(* CoDeSys 2.3.9.50 project: WTP_Pro_15_8_2016.pro *)
(* Libraries: STANDARD.LIB 5.6.98 12:03:02 *)

(* Task configuration *)
TASK Standard (PRIORITY := 0, INTERVAL := T#500ms);
	MAIN
END_TASK

(* Global variable list: Global_Variables *)
VAR_GLOBAL
	dummy: BOOL;
	GlobalON: TIME := T#5s;
	GlobalOFF: TIME := T#5s;
END_VAR

(* Data type *)
TYPE TEST :
STRUCT
	x : POINTER TO BOOL;
END_STRUCT
END_TYPE

(* Data type *)
TYPE TEST2 :
STRUCT
	X : BOOL;
END_STRUCT
END_TYPE

(* POU MAIN, ST *)
PROGRAM MAIN
VAR
	fbINLET_NEW_A: INLET_NEW_A;
	fbREUSE_WATER: REUSE_WATER;
END_VAR
STREAM_INLET_MIXER_1;
STREAM_INLET_MIXER_2;
INLET_SCREENING_OPERATION_2;
GRIT_REMOVAL_OPERATION;
SBR_TRANSFER_1;
SBR_TRANSFER_2;
REUSE_WATER_SYSTEM;
SBR_REACTOR_1;
SBR_REACTOR_2;
SLUDGE_THICKENING;

fbINLET_NEW_A();
fbREUSE_WATER();
END_PROGRAM

(* POU INLET_NEW_A, ST *)
FUNCTION_BLOCK INLET_NEW_A
VAR_INPUT
(*inlet*)
	i1: BOOL;
	i3: BOOL;
	i2: BOOL;
	i4: BOOL;

(*MIXER*)

	i5: BOOL;
	i6: BOOL;

(*penstock*)
	r1: BOOL; (*rs1*)
	i7: BOOL; (*ps open*)
	i8: BOOL;	(*ps open*)
	i10: BOOL;
	i9: BOOL;
	i11: BOOL;
	s1: BOOL;
	s2: BOOL;
	s3: BOOL;
	s4: BOOL;

(* sbr transfer *)
	i12: BOOL;
	i13: BOOL;


END_VAR
VAR_OUTPUT

(*inlet*)
	q1: BOOL;
	q2: BOOL;

(*MIXER*)

	q3: BOOL;
	q4: BOOL;

(*penstock*)
	q5: BOOL; (*ps1*)
	q6: BOOL; (*ps2*)
	q7: BOOL;
	q8: BOOL;
	q10: BOOL;
	q9: BOOL;
	q11: BOOL;
	q12: BOOL;
	q13: BOOL;
	q14: BOOL;
	q15: BOOL;
	q16: BOOL;
	q17: BOOL;
	q18: BOOL;
	q19: BOOL;
	q20: BOOL;
(* Grit Removal*)

	q21: BOOL;
	q22: BOOL;
	q23: BOOL;
	q24: BOOL;
	q25:BOOL;
	q26:BOOL;

(* sbr transfer *)

	q27: BOOL;
	q28: BOOL;

END_VAR
VAR
(*inlet*)
	m1: BOOL;
	ton1: TON;

(*MIXER*)


(*penstock*)
	penstock: INT;
	FailedGroupA: BOOL;
	FailedGroupB: BOOL;
	m2: BOOL;
	TP1: TP;
	m3: BOOL;
	TON2: TON;
	TON3: TON;
	TOF1: TOF;
	TON4 : TON;
	mr: BOOL;
	F_TRIG1: F_TRIG;
	R_TRIG1: R_TRIG;
	m4 : BOOL;
	TON5: TON;

END_VAR



(*
CASE penstock OF
0:
	q5 := TRUE;
	q6 := FALSE;
	IF FailedGroupA OR m2 THEN
		penstock := 1;
	END_IF
1 :
 	q6 := TRUE;
	IF FailedGroupB THEN
		penstock := 2;
	ELSIF i8 THEN
		penstock := 3;
	END_IF
2 :
	q5 := FALSE;
	q6 := FALSE;
	IF r1 THEN
		penstock := 0;
	END_IF
3:
	q6 := TRUE;
	q5 := FALSE;
	IF FailedGroupB OR m2 THEN
		penstock := 4;
	END_IF
4 :
	q6 := TRUE;
	IF FailedGroupA THEN
		penstock := 2;
	ELSIF i7 THEN
		penstock := 0;
	END_IF
END_CASE*)
(*EQ Pump*)
q1 := NOT i1 OR i3 OR m1;
q2 := i2 AND NOT i3 AND NOT m1;
ton1(IN:=i4 , PT:=t#5m , Q=>m1 , ET=> );

(*Mixer*)
q3 := NOT i5;
q4 := i6;


(*screen*)
FailedGroupA := s1 OR s2;
FailedGroupB := s3 OR s4;

m4 := ((NOT m4 AND (FailedGroupA OR m2)) OR m4) AND NOT((m4 AND (FailedGroupB OR m2)) OR r1);
q5 := (NOT m4 OR q5) AND NOT(( m4 AND i8) OR mr) ;
q6 := (m4 OR q6) AND NOT ((NOT m4 AND i7) OR mr);
mr := (mr OR (FailedGroupA AND FailedGroupB)) AND NOT r1;

TOF1(IN:=i11 , PT:=T#2m , Q=>i9 , ET=> );

F_TRIG1(CLK:=m4 );
R_TRIG1(CLK:=m4 );
TP1(IN:=(F_TRIG1.Q OR R_TRIG1.Q) , PT:= T#5m , Q=>m3 , ET=> );
m2 := i10 AND NOT m3;

TON4(IN:=NOT i9 OR NOT(q5 OR q6) , PT:=T#5m , Q=>q7 , ET=> );
TON2(IN:= i9 AND (q5 OR q6), PT := T#1h, Q=> q8);

TON3(IN:=q7,PT:=T#5m,Q=>q9);
q10 := q8;

q11 := q9;
q12 := q10;

q13 := NOT (i9 AND Q5);
q14 := (i9 AND Q5);

q15 := NOT(i9 AND q6);
q16 := (i9 AND q6);

q17 := q13;
q18 := q14;

q19 := q15;
q20 :=q18;

(*Grit Removal*)
q21 := i7;
q22 := i8;

q23 := NOT i9;
q24 := i9;

TON5(IN:= NOT i9, PT:=T#5m , Q=>q25 );
q26 := i9;


(*sbr transfer*)
q27  := NOT i12;
q28 := i13;
END_FUNCTION_BLOCK

(* POU REUSE_WATER, ST *)
FUNCTION_BLOCK REUSE_WATER
VAR_INPUT
	i3: BOOL;
	i1: BOOL;
	i4: BOOL;
	i2: BOOL;
	i5: BOOL;
	a1 : INT;
END_VAR
VAR_OUTPUT
	q1: BOOL;
	q2: BOOL;
	q3: BOOL;
	q4: BOOL;
	q5: BOOL;
	q6: BOOL;
	q7: BOOL;
	q8: BOOL;
	q9: BOOL;
END_VAR
VAR
	m1: BOOL;
	e1: BOOL;
	p1: REAL;
	TON1: TON;
	m2: BOOL;
END_VAR
p1 := INT_TO_REAL(a1) * (20.0/32767.0);

q1 := (p1 > 8) OR (NOT m1) OR e1 OR i3;
q2 := (p1 <= 6) AND m1;

q3:=(p1 > 6.4) OR (NOT m1) OR e1 OR i3;
q4 := (p1 <= 5.2) AND m1;

q5:=(p1 > 5.9) OR (NOT m1) OR e1 OR i3;
q6 := (p1 <= 4.7) AND m1;

TON1(IN:=((p1 < 3.5) AND m1) , PT:=T#5s , Q=>e1 , ET=> );
m2 := (i2 OR m2) AND i1;
m1 := i4 AND m2;

q7 := NOT i5 OR q7;
q8 := i5 AND q8;

q9 := TRUE;
END_FUNCTION_BLOCK

(* POU STREAM_INLET_MIXER_1, CFC *)
PROGRAM STREAM_INLET_MIXER_1
VAR
	LSL101A : inBlock;
	LSS101A : inBlock;
	LSH101A : inBlock;
	LSD101A : inBlock;
	LSL100A : inBlock;
	LSHL100A:inBlock;

	bCriticalEQFloatHi: BOOL;
	bWarningFloatSensorLow: BOOL;
	bCriticalFloatSensorDry: BOOL;



	EQPump_P101A_1_remote_mode AT%I* : BOOL;
	EQPump_P101A_1_overload AT%I* : BOOL;
	EQPump_P101A_1_incomplete AT%I* : BOOL;
	EQPump_P101A_1_status AT%I* : BOOL;

	EQPump_P101A_1_command AT%Q* : BOOL;

	EQPump_P101A_1_in : BOOL;
	EQPump_P101A_1_overload_error : BOOL;
	EQPump_P101A_1_incomplete_error : BOOL;
	EQPump_P101A_1_status_error : BOOL;
	EQPump_P101A_1_common_error : BOOL;
	EQPump_P101A_1_stop_error : BOOL;

	EQPump_P101A_1_overload_Filter : ErrorFilter;
	EQPump_P101A_1_incomplete_Filter : ErrorFilter;
	EQPump_P101A_1_status_Filter : ErrorFilter;
	EQPump_P101A_1_stop_Filter : ErrorFilter;



	EQPump_P101A_2_remote_mode AT%I* : BOOL;
	EQPump_P101A_2_overload AT%I* : BOOL;
	EQPump_P101A_2_incomplete AT%I* : BOOL;
	EQPump_P101A_2_status AT%I* : BOOL;

	EQPump_P101A_2_command AT%Q* : BOOL;

	EQPump_P101A_2_in : BOOL;
	EQPump_P101A_2_overload_error : BOOL;
	EQPump_P101A_2_incomplete_error : BOOL;
	EQPump_P101A_2_status_error : BOOL;
	EQPump_P101A_2_common_error : BOOL;
	EQPump_P101A_2_stop_error : BOOL;

	EQPump_P101A_2_overload_Filter : ErrorFilter;
	EQPump_P101A_2_incomplete_Filter : ErrorFilter;
	EQPump_P101A_2_status_Filter : ErrorFilter;
	EQPump_P101A_2_stop_Filter : ErrorFilter;

	EQPump_P101A_CriticalStartError : BOOL;

	Mixer_M101A_1_remote_mode AT%I* : BOOL;
	Mixer_M101A_1_overload AT%I* : BOOL;
	Mixer_M101A_1_incomplete AT%I* : BOOL;
	Mixer_M101A_1_status AT%I* : BOOL;

	Mixer_M101A_1_command AT%Q* : BOOL;

	Mixer_M101A_1_in : BOOL;
	Mixer_M101A_1_overload_error : BOOL;
	Mixer_M101A_1_incomplete_error : BOOL;
	Mixer_M101A_1_status_error : BOOL;
	Mixer_M101A_1_common_error : BOOL;
	Mixer_M101A_1_stop_error : BOOL;


	Mixer_M101A_1_overload_Filter : ErrorFilter;
	Mixer_M101A_1_incomplete_Filter : ErrorFilter;
	Mixer_M101A_1_status_Filter : ErrorFilter;
	Mixer_M101A_1_stop_Filter : ErrorFilter;


	Mixer_M101A_2_remote_mode AT%I* : BOOL;
	Mixer_M101A_2_overload AT%I* : BOOL;
	Mixer_M101A_2_incomplete AT%I* : BOOL;
	Mixer_M101A_2_status AT%I* : BOOL;

	Mixer_M101A_2_command AT%Q* : BOOL;

	Mixer_M101A_2_in : BOOL;
	Mixer_M101A_2_overload_error : BOOL;
	Mixer_M101A_2_incomplete_error : BOOL;
	Mixer_M101A_2_status_error : BOOL;
	Mixer_M101A_2_common_error : BOOL;
	Mixer_M101A_2_stop_error : BOOL;

	Mixer_M101A_2_overload_Filter : ErrorFilter;
	Mixer_M101A_2_incomplete_Filter : ErrorFilter;
	Mixer_M101A_2_status_Filter : ErrorFilter;
	Mixer_M101A_2_stop_Filter : ErrorFilter;

	Mixer_M101A_CriticalStartEror : BOOL;

	InletPump :Equipment_Dual;
	Mixer :Equipment_Dual;



END_VAR
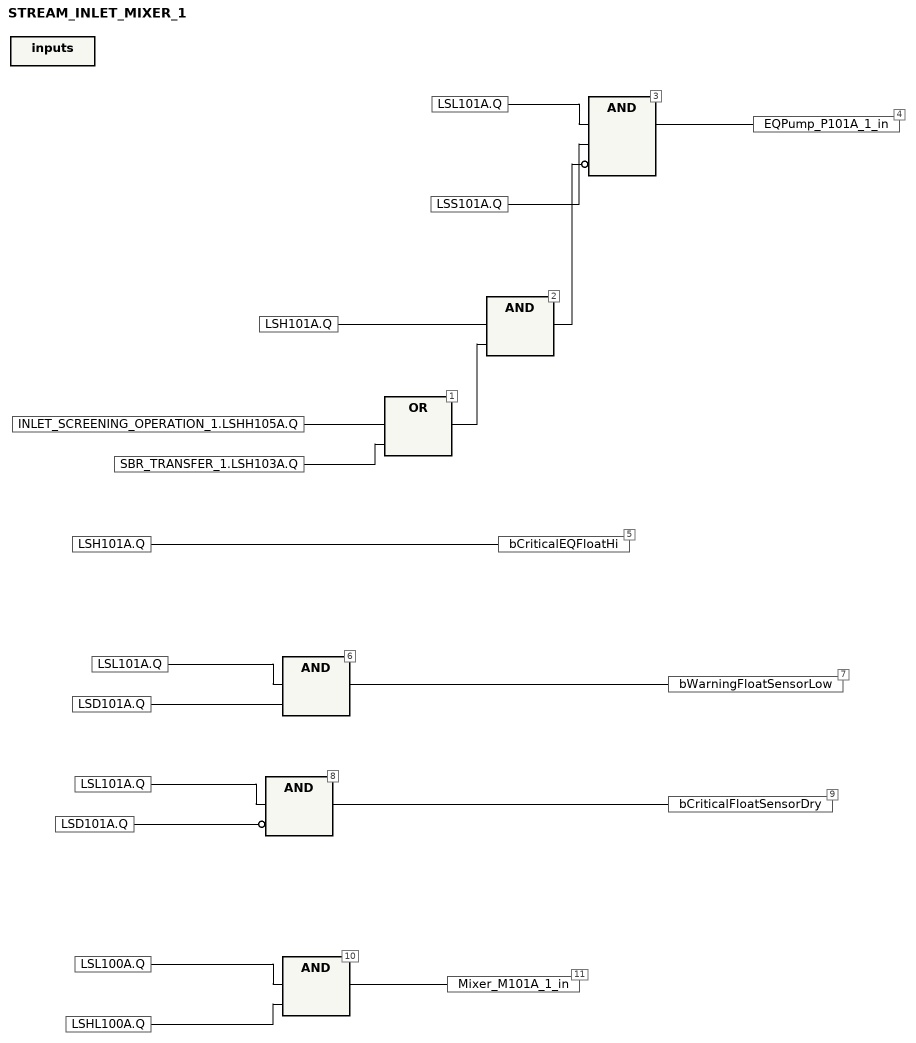
_CFC_ (* Continuous Function Chart, elements in execution order *)
#0 inputs()
#1 OR(INLET_SCREENING_OPERATION_1.LSHH105A.Q, SBR_TRANSFER_1.LSH103A.Q)
#2 AND(LSH101A.Q, #1)
#3 AND(LSL101A.Q, LSS101A.Q, NOT #2)
#4 EQPump_P101A_1_in <= #3
#5 bCriticalEQFloatHi <= LSH101A.Q
#6 AND(LSL101A.Q, LSD101A.Q)
#7 bWarningFloatSensorLow <= #6
#8 AND(LSL101A.Q, NOT LSD101A.Q)
#9 bCriticalFloatSensorDry <= #8
#10 AND(LSL100A.Q, LSHL100A.Q)
#11 Mixer_M101A_1_in <= #10
_END_CFC_
(* the same logic as Structured Text *)
inputs();
EQPump_P101A_1_in := LSL101A.Q AND LSS101A.Q AND NOT (LSH101A.Q AND (INLET_SCREENING_OPERATION_1.LSHH105A.Q OR SBR_TRANSFER_1.LSH103A.Q));
bCriticalEQFloatHi := LSH101A.Q;
bWarningFloatSensorLow := LSL101A.Q AND LSD101A.Q;
bCriticalFloatSensorDry := LSL101A.Q AND NOT LSD101A.Q;
Mixer_M101A_1_in := LSL100A.Q AND LSHL100A.Q;
END_PROGRAM
ACTION inputs:
	LSL101A();
	LSS101A();
	LSH101A();
	LSD101A();

	LSL100A();
	LSHL100A();



EQPump_P101A_1_overload_Filter(IN:=(EQPump_P101A_1_overload AND EQPump_P101A_1_in),PT:=T#10s,Q=>EQPump_P101A_1_overload_error);
EQPump_P101A_1_incomplete_Filter(IN:=(EQPump_P101A_1_incomplete AND EQPump_P101A_1_in),PT:=T#2s,Q=>EQPump_P101A_1_incomplete_error);
EQPump_P101A_1_status_Filter(IN:=(NOT EQPump_P101A_1_status AND EQPump_P101A_1_in),PT:=T#2s, Q=>EQPump_P101A_1_status_error);
EQPump_P101A_1_stop_Filter(IN:=( EQPump_P101A_1_status AND NOT EQPump_P101A_1_in),PT:=T#10s, Q=>EQPump_P101A_1_stop_error);

EQPump_P101A_1_common_error := EQPump_P101A_1_overload_error OR EQPump_P101A_1_incomplete_error OR EQPump_P101A_1_status_error OR EQPump_P101A_1_stop_error;



EQPump_P101A_2_overload_Filter(IN:=(EQPump_P101A_2_overload AND EQPump_P101A_2_in),PT:=T#10s,Q=>EQPump_P101A_2_overload_error);
EQPump_P101A_2_incomplete_Filter(IN:=(EQPump_P101A_2_incomplete AND EQPump_P101A_2_in),PT:=T#2s,Q=>EQPump_P101A_2_incomplete_error);
EQPump_P101A_2_status_Filter(IN:=(NOT EQPump_P101A_2_status AND EQPump_P101A_2_in),PT:=T#2s, Q=>EQPump_P101A_2_status_error);
EQPump_P101A_2_stop_Filter(IN:=( EQPump_P101A_2_status AND NOT EQPump_P101A_2_in),PT:=T#10s, Q=>EQPump_P101A_2_stop_error);

EQPump_P101A_2_common_error := EQPump_P101A_2_overload_error OR EQPump_P101A_2_incomplete_error OR EQPump_P101A_2_status_error OR EQPump_P101A_2_stop_error;

InletPump(
	ERROR1:=EQPump_P101A_1_common_error ,
	ERROR2:=EQPump_P101A_2_common_error ,
	IN1:=EQPump_P101A_1_in ,
	IN2:=EQPump_P101A_2_in ,
	remote1:=EQPump_P101A_1_remote_mode ,
	remote2:= EQPump_P101A_2_remote_mode,
	Command1=>EQPump_P101A_1_command ,
	Command2=>EQPump_P101A_2_command );


EQPump_P101A_CriticalStartError := EQPump_P101A_1_common_error AND EQPump_P101A_2_common_error;


Mixer_M101A_1_overload_Filter(IN:=(Mixer_M101A_1_overload AND Mixer_M101A_1_in),PT:=T#10s,Q=>Mixer_M101A_1_overload_error);
Mixer_M101A_1_incomplete_Filter(IN:=(Mixer_M101A_1_incomplete AND Mixer_M101A_1_in),PT:=T#2s,Q=>Mixer_M101A_1_incomplete_error);
Mixer_M101A_1_status_Filter(IN:=(NOT Mixer_M101A_1_status AND Mixer_M101A_1_in),PT:=T#2s, Q=>Mixer_M101A_1_status_error);
Mixer_M101A_1_stop_Filter(IN:=( Mixer_M101A_1_status AND NOT Mixer_M101A_1_in),PT:=T#10s, Q=>Mixer_M101A_1_stop_error);

Mixer_M101A_1_common_error := Mixer_M101A_1_overload_error OR Mixer_M101A_1_incomplete_error OR Mixer_M101A_1_status_error OR Mixer_M101A_1_stop_error;


Mixer_M101A_2_overload_Filter(IN:=(Mixer_M101A_2_overload AND Mixer_M101A_2_in),PT:=T#10s,Q=>Mixer_M101A_2_overload_error);
Mixer_M101A_2_incomplete_Filter(IN:=(Mixer_M101A_2_incomplete AND Mixer_M101A_2_in),PT:=T#2s,Q=>Mixer_M101A_2_incomplete_error);
Mixer_M101A_2_status_Filter(IN:=(NOT Mixer_M101A_2_status AND Mixer_M101A_2_in),PT:=T#2s, Q=>Mixer_M101A_2_status_error);
Mixer_M101A_2_stop_Filter(IN:=( Mixer_M101A_2_status AND NOT Mixer_M101A_2_in),PT:=T#10s, Q=>Mixer_M101A_2_stop_error);

Mixer_M101A_2_common_error := Mixer_M101A_2_overload_error OR Mixer_M101A_2_incomplete_error OR Mixer_M101A_2_status_error OR Mixer_M101A_2_stop_error;

Mixer(
	ERROR1:=Mixer_M101A_1_common_error ,
	ERROR2:=Mixer_M101A_2_common_error ,
	remote1:=Mixer_M101A_1_remote_mode ,
	remote2:= Mixer_M101A_2_remote_mode,
	IN1:=Mixer_M101A_1_in ,
	IN2:=Mixer_M101A_2_in ,
	Command1=>Mixer_M101A_1_command,
	Command2=>Mixer_M101A_2_command );

Mixer_M101A_CriticalStartEror := Mixer_M101A_1_common_error AND Mixer_M101A_2_common_error;
END_ACTION

(* POU module/inBlock, ST *)
FUNCTION_BLOCK inBlock
VAR_INPUT
END_VAR
VAR_OUTPUT
	Q : BOOL;
END_VAR
VAR
	IN AT%I* : BOOL;
	ON:TON;
	OFF: TON;
END_VAR
IF NOT Q THEN
	OFF(IN:= FALSE, PT:=GlobalOFF );
	ON(IN:= IN, PT:=GlobalON );
	IF ON.Q THEN
		ON(IN:= FALSE, PT:=GlobalON );
		Q:=TRUE;
	END_IF
ELSE
	ON(IN:= FALSE, PT:=GlobalON );
	OFF(IN:= NOT IN, PT:=GlobalOFF );
	IF OFF.Q THEN
		OFF(IN:= FALSE, PT:=GlobalON );
		Q:=FALSE;
	END_IF
END_IF
END_FUNCTION_BLOCK

(* POU module/ErrorFilter, ST *)
FUNCTION_BLOCK ErrorFilter
VAR_INPUT
	IN : BOOL;
	PT : TIME:=T#2s;
END_VAR
VAR_OUTPUT
	Q : BOOL;
END_VAR
VAR
	timer : TON;
END_VAR
IF PT <= T#0s THEN
	PT := T#2s;
END_IF

timer(IN:=IN , PT:=PT , Q=>Q );
END_FUNCTION_BLOCK

(* POU module/Equipment_Dual, ST *)
FUNCTION_BLOCK Equipment_Dual
VAR_INPUT
	ERROR1 : BOOL;
	ERROR2 : BOOL;
	remote1 : BOOL;
	remote2 : BOOL;
END_VAR
VAR_OUTPUT
	Command1 : BOOL;
	Command2 : BOOL;
END_VAR
VAR_IN_OUT
	IN1 : BOOL;
	IN2 : BOOL;
END_VAR
Command1 := IN1 AND remote1;
Command2 := IN2 AND remote2;
IN2 := ERROR1 AND remote2;
END_FUNCTION_BLOCK

(* POU INLET_SCREENING_OPERATION_1, CFC *)
PROGRAM INLET_SCREENING_OPERATION_1
VAR

	LSH105A : inBlock;
	LSHH105A: inBlock;
	Timer1: TON;
	StopTimer: TON;
	timerCompactor: TON;
	bFineScreenDual: BOOL;

	bWarningStreamLineOverflow: BOOL;


	Penstock_PS101A_1_status AT%I* : BOOL;
	Penstock_PS101A_1_command AT%Q* : BOOL;

	Penstock_PS101A_1_in : BOOL;
	Penstock_PS101A_1_open_error : BOOL;
	Penstock_PS101A_1_common_error : BOOL;
	Penstock_PS101A_1_close_error : BOOL;

	Penstock_PS101A_1_open_Filter : ErrorFilter;
	Penstock_PS101A_1_close_Filter : ErrorFilter;




	Penstock_PS101A_2_status AT%I* : BOOL;

	Penstock_PS101A_2_command AT%Q* : BOOL;

	Penstock_PS101A_2_in : BOOL;
	Penstock_PS101A_2_open_error : BOOL;
	Penstock_PS101A_2_common_error : BOOL;
	Penstock_PS101A_2_close_error : BOOL;

	Penstock_PS101A_2_open_Filter : ErrorFilter;
	Penstock_PS101A_2_close_Filter : ErrorFilter;


	Finescreen_F101A_1_remote_mode AT%I* : BOOL;
	Finescreen_F101A_1_overload AT%I* : BOOL;
	Finescreen_F101A_1_incomplete AT%I* : BOOL;
	Finescreen_F101A_1_status AT%I* : BOOL;

	Finescreen_F101A_1_command AT%Q* : BOOL;

	Finescreen_F101A_1_in : BOOL;
	Finescreen_F101A_1_overload_error : BOOL;
	Finescreen_F101A_1_incomplete_error : BOOL;
	Finescreen_F101A_1_status_error : BOOL;
	Finescreen_F101A_1_common_error : BOOL;
	Finescreen_F101A_1_stop_error : BOOL;

	Finescreen_F101A_1_overload_Filter : ErrorFilter;
	Finescreen_F101A_1_incomplete_Filter : ErrorFilter;
	Finescreen_F101A_1_status_Filter : ErrorFilter;
	Finescreen_F101A_1_stop_Filter : ErrorFilter;



	Finescreen_F101A_2_remote_mode AT%I* : BOOL;
	Finescreen_F101A_2_overload AT%I* : BOOL;
	Finescreen_F101A_2_incomplete AT%I* : BOOL;
	Finescreen_F101A_2_status AT%I* : BOOL;

	Finescreen_F101A_2_command AT%Q* : BOOL;

	Finescreen_F101A_2_in : BOOL;
	Finescreen_F101A_2_overload_error : BOOL;
	Finescreen_F101A_2_incomplete_error : BOOL;
	Finescreen_F101A_2_status_error : BOOL;
	Finescreen_F101A_2_common_error : BOOL;
	Finescreen_F101A_2_stop_error : BOOL;

	Finescreen_F101A_2_overload_Filter : ErrorFilter;
	Finescreen_F101A_2_incomplete_Filter : ErrorFilter;
	Finescreen_F101A_2_status_Filter : ErrorFilter;
	Finescreen_F101A_2_stop_Filter : ErrorFilter;

	FineScreen :Equipment_Dual;


	WaterSprayScreen_XV101A_1_open_status AT%I* : BOOL;
	WaterSprayScreen_XV101A_1_close_status AT%I* : BOOL;

	WaterSprayScreen_XV101A_1_command AT%Q* : BOOL;

	WaterSprayScreen_XV101A_1_in : BOOL;
	WaterSprayScreen_XV101A_1_open_error : BOOL;
	WaterSprayScreen_XV101A_1_common_error : BOOL;
	WaterSprayScreen_XV101A_1_close_error : BOOL;

	WaterSprayScreen_XV101A_1_open_Filter : ErrorFilter;
	WaterSprayScreen_XV101A_1_close_Filter : ErrorFilter;



	WaterSprayScreen_XV101A_2_open_status AT%I* : BOOL;
	WaterSprayScreen_XV101A_2_close_status AT%I* : BOOL;

	WaterSprayScreen_XV101A_2_command AT%Q* : BOOL;

	WaterSprayScreen_XV101A_2_in : BOOL;
	WaterSprayScreen_XV101A_2_open_error : BOOL;
	WaterSprayScreen_XV101A_2_common_error : BOOL;
	WaterSprayScreen_XV101A_2_close_error : BOOL;

	WaterSprayScreen_XV101A_2_open_Filter : ErrorFilter;
	WaterSprayScreen_XV101A_2_close_Filter : ErrorFilter;




	WaterSprayScreen1: Equipment_Timed;
	WaterSprayScreen2: Equipment_Timed;



	ScrewConveyer_C102A_remote_mode AT%I* : BOOL;
	ScrewConveyer_C102A_overload AT%I* : BOOL;
	ScrewConveyer_C102A_incomplete AT%I* : BOOL;
	ScrewConveyer_C102A_status AT%I* : BOOL;

	ScrewConveyer_C102A_command AT%Q* : BOOL;

	ScrewConveyer_C102A_in : BOOL;
	ScrewConveyer_C102A_overload_error : BOOL;
	ScrewConveyer_C102A_incomplete_error : BOOL;
	ScrewConveyer_C102A_status_error : BOOL;
	ScrewConveyer_C102A_common_error : BOOL;
	ScrewConveyer_C102A_stop_error : BOOL;

	ScrewConveyer_C102A_overload_Filter : ErrorFilter;
	ScrewConveyer_C102A_incomplete_Filter : ErrorFilter;
	ScrewConveyer_C102A_status_Filter : ErrorFilter;
	ScrewConveyer_C102A_stop_Filter : ErrorFilter;

	ScreenCompactor_C101A_remote_mode AT%I* : BOOL;
	ScreenCompactor_C101A_overload AT%I* : BOOL;
	ScreenCompactor_C101A_incomplete AT%I* : BOOL;
	ScreenCompactor_C101A_status AT%I* : BOOL;

	ScreenCompactor_C101A_command AT%Q* : BOOL;

	ScreenCompactor_C101A_in : BOOL;
	ScreenCompactor_C101A_overload_error : BOOL;
	ScreenCompactor_C101A_incomplete_error : BOOL;
	ScreenCompactor_C101A_status_error : BOOL;
	ScreenCompactor_C101A_common_error : BOOL;
	ScreenCompactor_C101A_stop_error : BOOL;

	ScreenCompactor_C101A_overload_Filter : ErrorFilter;
	ScreenCompactor_C101A_incomplete_Filter : ErrorFilter;
	ScreenCompactor_C101A_status_Filter : ErrorFilter;
	ScreenCompactor_C101A_stop_Filter : ErrorFilter;

	ContinuousWaterSpray_XV102A_remote_mode AT%I* : BOOL;
	ContinuousWaterSpray_XV102A_overload AT%I* : BOOL;
	ContinuousWaterSpray_XV102A_incomplete AT%I* : BOOL;
	ContinuousWaterSpray_XV102A_status AT%I* : BOOL;

	ContinuousWaterSpray_XV102A_command AT%Q* : BOOL;

	ContinuousWaterSpray_XV102A_in : BOOL;
	ContinuousWaterSpray_XV102A_overload_error : BOOL;
	ContinuousWaterSpray_XV102A_incomplete_error : BOOL;
	ContinuousWaterSpray_XV102A_status_error : BOOL;
	ContinuousWaterSpray_XV102A_common_error : BOOL;
	ContinuousWaterSpray_XV102A_stop_error : BOOL;

	ContinuousWaterSpray_XV102A_overload_Filter : ErrorFilter;
	ContinuousWaterSpray_XV102A_incomplete_Filter : ErrorFilter;
	ContinuousWaterSpray_XV102A_status_Filter : ErrorFilter;
	ContinuousWaterSpray_XV102A_stop_Filter : ErrorFilter;

	WaterSprayOff1: TOF;
	WaterSprayOff2: TOF;
END_VAR
VAR (* helpers for the ST form of the networks *)
	_en57 : BOOL;
	_t57 : BOOL;
	_en85 : BOOL;
	_t85 : BOOL;
END_VAR
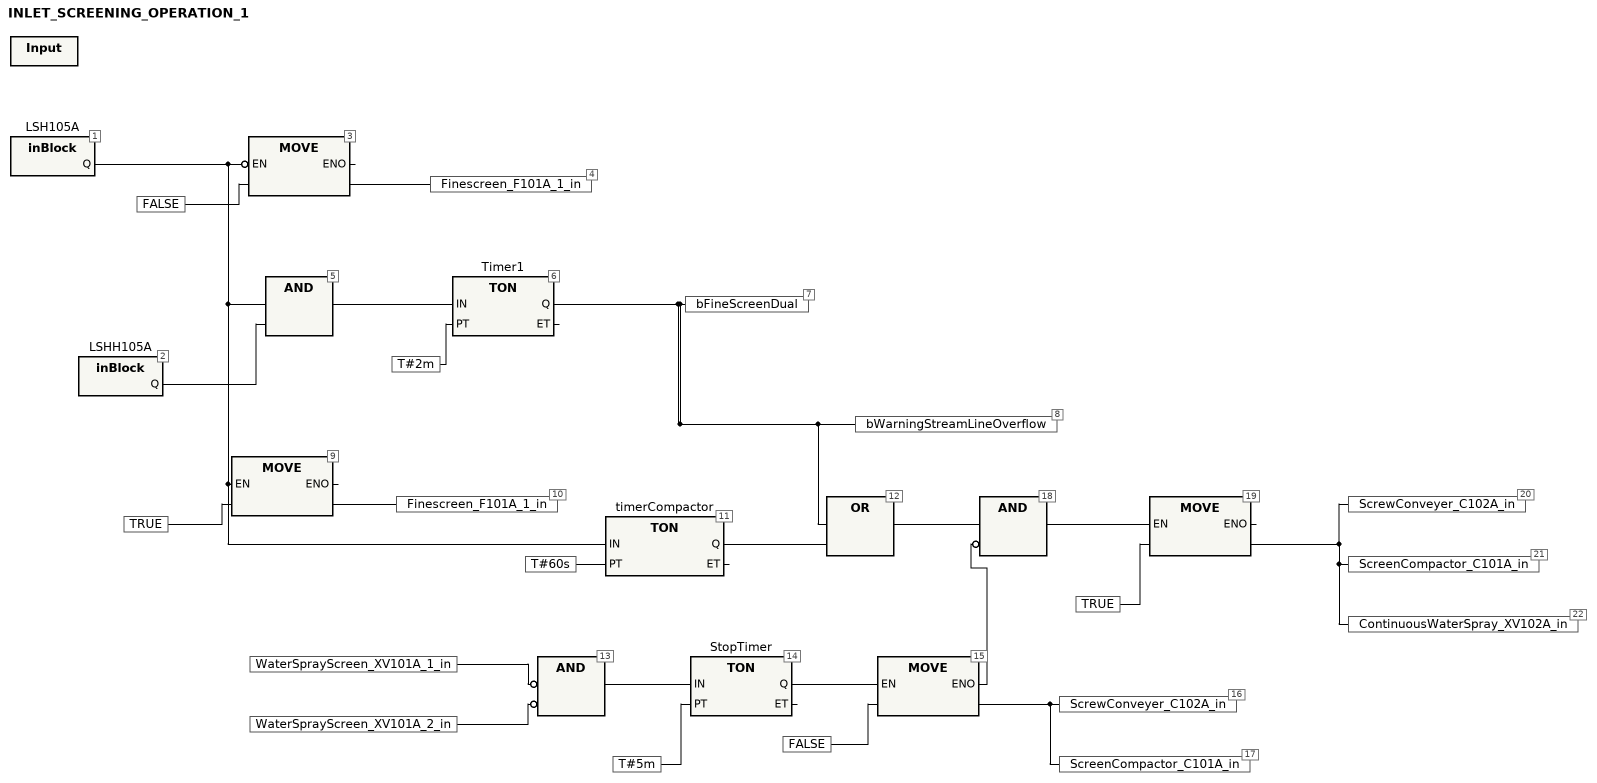
_CFC_ (* Continuous Function Chart, elements in execution order *)
#0 Input()
#1 LSH105A:inBlock()
#2 LSHH105A:inBlock()
#3 MOVE(EN: NOT #1.Q, FALSE)
#4 Finescreen_F101A_1_in <= #3
#5 AND(#1.Q, #2.Q)
#6 Timer1:TON(IN: #5, PT: T#2m)
#7 bFineScreenDual <= #6.Q
#8 bWarningStreamLineOverflow <= #6.Q
#9 MOVE(EN: #1.Q, TRUE)
#10 Finescreen_F101A_1_in <= #9
#11 timerCompactor:TON(IN: #1.Q, PT: T#60s)
#12 OR(#6.Q, #11.Q)
#13 AND(NOT WaterSprayScreen_XV101A_1_in, NOT WaterSprayScreen_XV101A_2_in)
#14 StopTimer:TON(IN: #13, PT: T#5m)
#15 MOVE(EN: #14.Q, FALSE)
#16 ScrewConveyer_C102A_in <= #15
#17 ScreenCompactor_C101A_in <= #15
#18 AND(#12, NOT #15.ENO)
#19 MOVE(EN: #18, TRUE)
#20 ScrewConveyer_C102A_in <= #19
#21 ScreenCompactor_C101A_in <= #19
#22 ContinuousWaterSpray_XV102A_in <= #19
_END_CFC_
(* the same logic as Structured Text *)
Input();
LSH105A();
LSHH105A();
IF NOT LSH105A.Q THEN Finescreen_F101A_1_in := FALSE; END_IF;
Timer1(IN := LSH105A.Q AND LSHH105A.Q, PT := T#2m);
bFineScreenDual := Timer1.Q;
bWarningStreamLineOverflow := Timer1.Q;
IF LSH105A.Q THEN Finescreen_F101A_1_in := TRUE; END_IF;
timerCompactor(IN := LSH105A.Q, PT := T#60s);
StopTimer(IN := NOT WaterSprayScreen_XV101A_1_in AND NOT WaterSprayScreen_XV101A_2_in, PT := T#5m);
_en57 := StopTimer.Q;
IF _en57 THEN _t57 := FALSE; END_IF;
IF _en57 THEN ScrewConveyer_C102A_in := _t57; END_IF;
IF _en57 THEN ScreenCompactor_C101A_in := _t57; END_IF;
_en85 := (Timer1.Q OR timerCompactor.Q) AND NOT _en57;
IF _en85 THEN _t85 := TRUE; END_IF;
IF _en85 THEN ScrewConveyer_C102A_in := _t85; END_IF;
IF _en85 THEN ScreenCompactor_C101A_in := _t85; END_IF;
IF _en85 THEN ContinuousWaterSpray_XV102A_in := _t85; END_IF;
END_PROGRAM
ACTION Input:
LSH105A( );
LSHH105A( );

Penstock_PS101A_1_command := Penstock_PS101A_1_in;
Penstock_PS101A_1_open_Filter(IN:=(NOT Penstock_PS101A_1_status AND Penstock_PS101A_1_in),PT:=T#10s, Q=>Penstock_PS101A_1_open_error);
Penstock_PS101A_1_close_Filter(IN:=( Penstock_PS101A_1_status AND NOT Penstock_PS101A_1_in),PT:=T#10s, Q=>Penstock_PS101A_1_close_error);

Penstock_PS101A_1_common_error := Penstock_PS101A_1_open_error OR Penstock_PS101A_1_close_error;


Penstock_PS101A_2_command := Penstock_PS101A_2_in;
Penstock_PS101A_2_open_Filter(IN:=(NOT Penstock_PS101A_2_status AND Penstock_PS101A_2_in),PT:=T#10s, Q=>Penstock_PS101A_2_open_error);
Penstock_PS101A_2_close_Filter(IN:=( Penstock_PS101A_2_status AND NOT Penstock_PS101A_2_in),PT:=T#10s, Q=>Penstock_PS101A_2_close_error);

Penstock_PS101A_2_common_error := Penstock_PS101A_2_open_error OR Penstock_PS101A_2_close_error;




Finescreen_F101A_1_overload_Filter(IN:=(Finescreen_F101A_1_overload AND Finescreen_F101A_1_in),PT:=T#2s,Q=>Finescreen_F101A_1_overload_error);
Finescreen_F101A_1_incomplete_Filter(IN:=(Finescreen_F101A_1_incomplete AND Finescreen_F101A_1_in),PT:=T#2s,Q=>Finescreen_F101A_1_incomplete_error);
Finescreen_F101A_1_status_Filter(IN:=(NOT Finescreen_F101A_1_status AND Finescreen_F101A_1_in),PT:=T#10s, Q=>Finescreen_F101A_1_status_error);
Finescreen_F101A_1_stop_Filter(IN:=( Finescreen_F101A_1_status AND NOT Finescreen_F101A_1_in),PT:=T#10s, Q=>Finescreen_F101A_1_stop_error);

Finescreen_F101A_1_common_error := Finescreen_F101A_1_overload_error OR Finescreen_F101A_1_incomplete_error OR Finescreen_F101A_1_status_error OR Finescreen_F101A_1_stop_error;


Finescreen_F101A_2_overload_Filter(IN:=(Finescreen_F101A_2_overload AND Finescreen_F101A_2_in),PT:=T#2s,Q=>Finescreen_F101A_2_overload_error);
Finescreen_F101A_2_incomplete_Filter(IN:=(Finescreen_F101A_2_incomplete AND Finescreen_F101A_2_in),PT:=T#2s,Q=>Finescreen_F101A_2_incomplete_error);
Finescreen_F101A_2_status_Filter(IN:=(NOT Finescreen_F101A_2_status AND Finescreen_F101A_2_in),PT:=T#10s, Q=>Finescreen_F101A_2_status_error);
Finescreen_F101A_2_stop_Filter(IN:=( Finescreen_F101A_2_status AND NOT Finescreen_F101A_2_in),PT:=T#10s, Q=>Finescreen_F101A_2_stop_error);

Finescreen_F101A_2_common_error := Finescreen_F101A_2_overload_error OR Finescreen_F101A_2_incomplete_error OR Finescreen_F101A_2_status_error OR Finescreen_F101A_2_stop_error;


FineScreen(
	ERROR1:=Finescreen_F101A_1_common_error ,
	ERROR2:=Finescreen_F101A_2_common_error ,
	IN1:= Finescreen_F101A_1_in,
	IN2:=Finescreen_F101A_2_in ,
	remote1:=Finescreen_F101A_1_remote_mode ,
	remote2:= Finescreen_F101A_2_remote_mode,
	Command1=>Finescreen_F101A_1_command ,
	Command2=>Finescreen_F101A_2_command );

IF bFineScreenDual THEN
	Finescreen_F101A_2_command := TRUE;
END_IF


Penstock_PS101A_1_in := Finescreen_F101A_1_command;
Penstock_PS101A_2_in := Finescreen_F101A_2_command;

WaterSprayOff1(IN:=Finescreen_F101A_1_command , PT:=T#2m , Q=>WaterSprayScreen_XV101A_1_in , ET=> );
WaterSprayOff2(IN:=Finescreen_F101A_2_command , PT:=T#2m , Q=>WaterSprayScreen_XV101A_2_in , ET=> );


WaterSprayScreen1(
	PT1:= T#1m,
	PT2:= T#5m,
	IN1:= WaterSprayScreen_XV101A_1_in,
	Command1=>WaterSprayScreen_XV101A_1_command );

WaterSprayScreen_XV101A_1_open_Filter(IN:=((NOT WaterSprayScreen_XV101A_1_open_status OR WaterSprayScreen_XV101A_1_close_status) AND WaterSprayScreen_XV101A_1_command),PT:=T#10s, Q=>WaterSprayScreen_XV101A_1_open_error);
WaterSprayScreen_XV101A_1_close_Filter(IN:=(( WaterSprayScreen_XV101A_1_open_status OR NOT WaterSprayScreen_XV101A_1_close_status) AND NOT WaterSprayScreen_XV101A_1_command),PT:=T#10s, Q=>WaterSprayScreen_XV101A_1_close_error);

WaterSprayScreen_XV101A_1_common_error := WaterSprayScreen_XV101A_1_open_error OR WaterSprayScreen_XV101A_1_close_error;


WaterSprayScreen2(
	PT1:= T#1m,
	PT2:= T#5m,
	IN1:= WaterSprayScreen_XV101A_2_in,
	Command1=>WaterSprayScreen_XV101A_2_command );

WaterSprayScreen_XV101A_2_open_Filter(IN:=((NOT WaterSprayScreen_XV101A_2_open_status OR WaterSprayScreen_XV101A_2_close_status) AND WaterSprayScreen_XV101A_2_in),PT:=T#10s, Q=>WaterSprayScreen_XV101A_2_open_error);
WaterSprayScreen_XV101A_2_close_Filter(IN:=((WaterSprayScreen_XV101A_2_open_status OR NOT WaterSprayScreen_XV101A_2_close_status) AND NOT WaterSprayScreen_XV101A_2_in),PT:=T#10s, Q=>WaterSprayScreen_XV101A_2_close_error);

WaterSprayScreen_XV101A_2_common_error := WaterSprayScreen_XV101A_2_open_error OR WaterSprayScreen_XV101A_2_close_error;


ScrewConveyer_C102A_command :=ScrewConveyer_C102A_in AND ScrewConveyer_C102A_remote_mode;
ScrewConveyer_C102A_overload_Filter(IN:=(ScrewConveyer_C102A_overload AND ScrewConveyer_C102A_in),PT:=T#2s,Q=>ScrewConveyer_C102A_overload_error);
ScrewConveyer_C102A_incomplete_Filter(IN:=(ScrewConveyer_C102A_incomplete AND ScrewConveyer_C102A_in),PT:=T#2s,Q=>ScrewConveyer_C102A_incomplete_error);
ScrewConveyer_C102A_status_Filter(IN:=(NOT ScrewConveyer_C102A_status AND ScrewConveyer_C102A_in),PT:=T#10s, Q=>ScrewConveyer_C102A_status_error);
ScrewConveyer_C102A_stop_Filter(IN:=( ScrewConveyer_C102A_status AND NOT ScrewConveyer_C102A_in),PT:=T#10s, Q=>ScrewConveyer_C102A_stop_error);

ScrewConveyer_C102A_common_error := ScrewConveyer_C102A_overload_error OR ScrewConveyer_C102A_incomplete_error OR ScrewConveyer_C102A_status_error OR ScrewConveyer_C102A_stop_error;


ScreenCompactor_C101A_command := ScreenCompactor_C101A_in OR ScreenCompactor_C101A_remote_mode;
ScreenCompactor_C101A_overload_Filter(IN:=(ScreenCompactor_C101A_overload AND ScreenCompactor_C101A_in),PT:=T#2s,Q=>ScreenCompactor_C101A_overload_error);
ScreenCompactor_C101A_incomplete_Filter(IN:=(ScreenCompactor_C101A_incomplete AND ScreenCompactor_C101A_in),PT:=T#2s,Q=>ScreenCompactor_C101A_incomplete_error);
ScreenCompactor_C101A_status_Filter(IN:=(NOT ScreenCompactor_C101A_status AND ScreenCompactor_C101A_in),PT:=T#10s, Q=>ScreenCompactor_C101A_status_error);
ScreenCompactor_C101A_stop_Filter(IN:=( ScreenCompactor_C101A_status AND NOT ScreenCompactor_C101A_in),PT:=T#10s, Q=>ScreenCompactor_C101A_stop_error);

ScreenCompactor_C101A_common_error := ScreenCompactor_C101A_overload_error OR ScreenCompactor_C101A_incomplete_error OR ScreenCompactor_C101A_status_error OR ScreenCompactor_C101A_stop_error;


ContinuousWaterSpray_XV102A_command := ContinuousWaterSpray_XV102A_in;
ContinuousWaterSpray_XV102A_overload_Filter(IN:=(ContinuousWaterSpray_XV102A_overload AND ContinuousWaterSpray_XV102A_in),PT:=T#2s,Q=>ContinuousWaterSpray_XV102A_overload_error);
ContinuousWaterSpray_XV102A_incomplete_Filter(IN:=(ContinuousWaterSpray_XV102A_incomplete AND ContinuousWaterSpray_XV102A_in),PT:=T#2s,Q=>ContinuousWaterSpray_XV102A_incomplete_error);
ContinuousWaterSpray_XV102A_status_Filter(IN:=(NOT ContinuousWaterSpray_XV102A_status AND ContinuousWaterSpray_XV102A_in),PT:=T#10s, Q=>ContinuousWaterSpray_XV102A_status_error);
ContinuousWaterSpray_XV102A_stop_Filter(IN:=( ContinuousWaterSpray_XV102A_status AND NOT ContinuousWaterSpray_XV102A_in),PT:=T#10s, Q=>ContinuousWaterSpray_XV102A_stop_error);

ContinuousWaterSpray_XV102A_common_error := ContinuousWaterSpray_XV102A_overload_error OR ContinuousWaterSpray_XV102A_incomplete_error OR ContinuousWaterSpray_XV102A_status_error OR ContinuousWaterSpray_XV102A_stop_error;
END_ACTION

(* POU module/Equipment_Timed, ST *)
FUNCTION_BLOCK Equipment_Timed
VAR_INPUT
	PT1 : TIME;
	PT2 : TIME;
END_VAR
VAR_OUTPUT
	Command1 : BOOL;
END_VAR
VAR_IN_OUT
	IN1 : BOOL;
END_VAR
VAR
	timer1: TON;
	timer2: TON;
END_VAR
timer1(IN:=NOT timer2.Q AND IN1 , PT:=PT1 , Q=> , ET=> );
timer2(IN:=timer1.Q , PT:=PT2 , Q=> , ET=> );

command1 := IN1 AND NOT timer1.Q;
END_FUNCTION_BLOCK

(* POU SBR_TRANSFER_1, CFC *)
PROGRAM SBR_TRANSFER_1
VAR
	LSL103A : inBlock;
	LSS103A : inBlock;
	LSH103A : inBlock;
	LSD103A : inBlock;


	bWarningSBRDry: BOOL;
	bCriticalSBRDry: BOOL;
	bCriticalSBRHi: BOOL;

	SBRTransferPump_P102A_1_remote_mode AT%I* : BOOL;
	SBRTransferPump_P102A_1_overload AT%I* : BOOL;
	SBRTransferPump_P102A_1_incomplete AT%I* : BOOL;
	SBRTransferPump_P102A_1_status AT%I* : BOOL;

	SBRTransferPump_P102A_1_command AT%Q* : BOOL;

	SBRTransferPump_P102A_1_in : BOOL;
	SBRTransferPump_P102A_1_overload_error : BOOL;
	SBRTransferPump_P102A_1_incomplete_error : BOOL;
	SBRTransferPump_P102A_1_status_error : BOOL;
	SBRTransferPump_P102A_1_common_error : BOOL;
	SBRTransferPump_P102A_1_stop_error : BOOL;

	SBRTransferPump_P102A_1_overload_Filter : ErrorFilter;
	SBRTransferPump_P102A_1_incomplete_Filter : ErrorFilter;
	SBRTransferPump_P102A_1_status_Filter : ErrorFilter;
	SBRTransferPump_P102A_1_stop_Filter : ErrorFilter;



	SBRTransferPump_P102A_2_remote_mode AT%I* : BOOL;
	SBRTransferPump_P102A_2_overload AT%I* : BOOL;
	SBRTransferPump_P102A_2_incomplete AT%I* : BOOL;
	SBRTransferPump_P102A_2_status AT%I* : BOOL;

	SBRTransferPump_P102A_2_command AT%Q* : BOOL;

	SBRTransferPump_P102A_2_in : BOOL;
	SBRTransferPump_P102A_2_overload_error : BOOL;
	SBRTransferPump_P102A_2_incomplete_error : BOOL;
	SBRTransferPump_P102A_2_status_error : BOOL;
	SBRTransferPump_P102A_2_common_error : BOOL;
	SBRTransferPump_P102A_2_stop_error : BOOL;

	SBRTransferPump_P102A_2_overload_Filter : ErrorFilter;
	SBRTransferPump_P102A_2_incomplete_Filter : ErrorFilter;
	SBRTransferPump_P102A_2_status_Filter : ErrorFilter;
	SBRTransferPump_P102A_2_stop_Filter : ErrorFilter;
	SBRTransferPump_P102A_CriticalStartingError: BOOL;
	SBRTransferPump_P102A: Equipment_Dual;
END_VAR
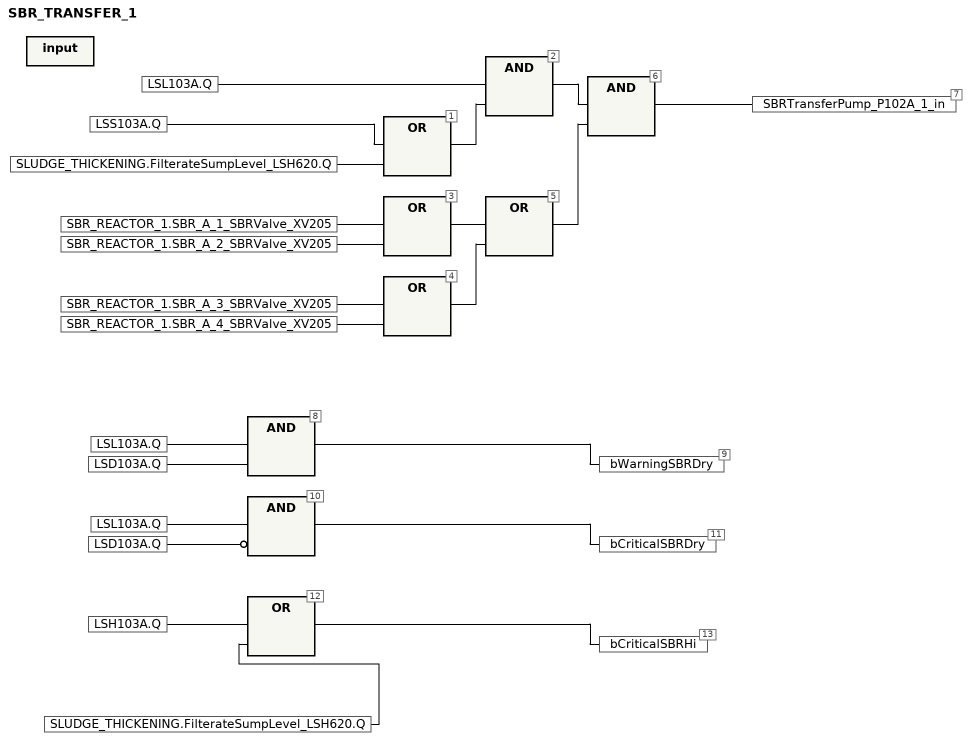
_CFC_ (* Continuous Function Chart, elements in execution order *)
#0 input()
#1 OR(LSS103A.Q, SLUDGE_THICKENING.FilterateSumpLevel_LSH620.Q)
#2 AND(LSL103A.Q, #1)
#3 OR(SBR_REACTOR_1.SBR_A_1_SBRValve_XV205, SBR_REACTOR_1.SBR_A_2_SBRValve_XV205)
#4 OR(SBR_REACTOR_1.SBR_A_3_SBRValve_XV205, SBR_REACTOR_1.SBR_A_4_SBRValve_XV205)
#5 OR(#3, #4)
#6 AND(#2, #5)
#7 SBRTransferPump_P102A_1_in <= #6
#8 AND(LSL103A.Q, LSD103A.Q)
#9 bWarningSBRDry <= #8
#10 AND(LSL103A.Q, NOT LSD103A.Q)
#11 bCriticalSBRDry <= #10
#12 OR(LSH103A.Q, SLUDGE_THICKENING.FilterateSumpLevel_LSH620.Q)
#13 bCriticalSBRHi <= #12
_END_CFC_
(* the same logic as Structured Text *)
input();
SBRTransferPump_P102A_1_in := (LSL103A.Q AND (LSS103A.Q OR SLUDGE_THICKENING.FilterateSumpLevel_LSH620.Q)) AND ((SBR_REACTOR_1.SBR_A_1_SBRValve_XV205 OR SBR_REACTOR_1.SBR_A_2_SBRValve_XV205) OR (SBR_REACTOR_1.SBR_A_3_SBRValve_XV205 OR SBR_REACTOR_1.SBR_A_4_SBRValve_XV205));
bWarningSBRDry := LSL103A.Q AND LSD103A.Q;
bCriticalSBRDry := LSL103A.Q AND NOT LSD103A.Q;
bCriticalSBRHi := LSH103A.Q OR SLUDGE_THICKENING.FilterateSumpLevel_LSH620.Q;
END_PROGRAM
ACTION Input:
LSD103A( );
LSH103A();
LSL103A( );
LSS103A( );


SBRTransferPump_P102A_1_overload_Filter(IN:=(SBRTransferPump_P102A_1_overload AND SBRTransferPump_P102A_1_in),PT:=T#2s,Q=>SBRTransferPump_P102A_1_overload_error);
SBRTransferPump_P102A_1_incomplete_Filter(IN:=(SBRTransferPump_P102A_1_incomplete AND SBRTransferPump_P102A_1_in),PT:=T#2s,Q=>SBRTransferPump_P102A_1_incomplete_error);
SBRTransferPump_P102A_1_status_Filter(IN:=(NOT SBRTransferPump_P102A_1_status AND SBRTransferPump_P102A_1_in),PT:=T#10s, Q=>SBRTransferPump_P102A_1_status_error);
SBRTransferPump_P102A_1_stop_Filter(IN:=( SBRTransferPump_P102A_1_status AND NOT SBRTransferPump_P102A_1_in),PT:=T#10s, Q=>SBRTransferPump_P102A_1_stop_error);

SBRTransferPump_P102A_1_common_error := SBRTransferPump_P102A_1_overload_error OR SBRTransferPump_P102A_1_incomplete_error OR SBRTransferPump_P102A_1_status_error OR SBRTransferPump_P102A_1_stop_error;


SBRTransferPump_P102A_2_overload_Filter(IN:=(SBRTransferPump_P102A_2_overload AND SBRTransferPump_P102A_2_in),PT:=T#2s,Q=>SBRTransferPump_P102A_2_overload_error);
SBRTransferPump_P102A_2_incomplete_Filter(IN:=(SBRTransferPump_P102A_2_incomplete AND SBRTransferPump_P102A_2_in),PT:=T#2s,Q=>SBRTransferPump_P102A_2_incomplete_error);
SBRTransferPump_P102A_2_status_Filter(IN:=(NOT SBRTransferPump_P102A_2_status AND SBRTransferPump_P102A_2_in),PT:=T#10s, Q=>SBRTransferPump_P102A_2_status_error);
SBRTransferPump_P102A_2_stop_Filter(IN:=( SBRTransferPump_P102A_2_status AND NOT SBRTransferPump_P102A_2_in),PT:=T#10s, Q=>SBRTransferPump_P102A_2_stop_error);

SBRTransferPump_P102A_2_common_error := SBRTransferPump_P102A_2_overload_error OR SBRTransferPump_P102A_2_incomplete_error OR SBRTransferPump_P102A_2_status_error OR SBRTransferPump_P102A_2_stop_error;

SBRTransferPump_P102A_CriticalStartingError := SBRTransferPump_P102A_1_common_error AND SBRTransferPump_P102A_2_common_error;

SBRTransferPump_P102A(
	ERROR1:=SBRTransferPump_P102A_1_common_error ,
	ERROR2:=SBRTransferPump_P102A_2_common_error ,
	remote1:=SBRTransferPump_P102A_1_remote_mode ,
	remote2:=SBRTransferPump_P102A_2_remote_mode ,
	IN1:= SBRTransferPump_P102A_1_in,
	IN2:=SBRTransferPump_P102A_2_in ,
	Command1=>SBRTransferPump_P102A_1_command ,
	Command2=>SBRTransferPump_P102A_2_command );
END_ACTION

(* POU SLUDGE_THICKENING, CFC *)
PROGRAM SLUDGE_THICKENING
VAR
	SludgeTankLevel_LSH501A: inBlock;
	SludgeTankLevel_LSH501B: inBlock;
	SludgeTankLevel_LSL501A: inBlock;
	SludgeTankLevel_LSL501B: inBlock;
	SludgePitSensor_LSH600: inBlock;
	PolimerTank_LSLPU501: inBlock;
	PolimerTank_LSHPU501: inBlock;
	FilterateSumpLevel_LSL620: inBlock;
	FilterateSumpLevel_LSH620: inBlock;

	PressureSwitch_PSL505A AT%I*: BOOL;
	PressureSwitch_PSL505B AT%I*: BOOL;

	PolimerValveOpen_XVPU501A AT%Q*: BOOL;
	PolimerValveClose_XVPU501A AT%Q*: BOOL;
	PolimerValveOpen_XVPU501B AT%Q*: BOOL;
	PolimerValveClose_XVPU501B AT%Q*: BOOL;
	DiagramValvaOpen_XVPU502 AT%Q*: BOOL;
	SolenoidValve_XV505A AT%Q*: BOOL;
	SolenoidValve_XV505B AT%Q*: BOOL;
	BlowerValve_XV501A	AT%Q* : BOOL;
	BlowerValve_XV501B AT%Q* : BOOL;


	bWarning_PolimerLow: BOOL;


	Blower_P505: BOOL;
	SludgeFeedPump_P501: BOOL;
	DrumThickener_D503: BOOL;
	BackWashWaterPump: BOOL;
	bFloculator_M502A: BOOL;
	bFloculator_M502B: BOOL;

	StreamA_Failed: BOOL;
	StreamB_Failed: BOOL;
	DrumThickenerError: BOOL;
	FluoculatorError: BOOL;
	BackwashFailed: BOOL;
	bDolanError: BOOL;

	PolymerTimer: TON;

	FilteratePump_P602_A_remote_mode AT%I* : BOOL;
	FilteratePump_P602_A_overload AT%I* : BOOL;
	FilteratePump_P602_A_incomplete AT%I* : BOOL;
	FilteratePump_P602_A_status AT%I* : BOOL;

	FilteratePump_P602_A_command AT%Q* : BOOL;

	FilteratePump_P602_A_in : BOOL;
	FilteratePump_P602_A_overload_error : BOOL;
	FilteratePump_P602_A_incomplete_error : BOOL;
	FilteratePump_P602_A_status_error : BOOL;
	FilteratePump_P602_A_common_error : BOOL;
	FilteratePump_P602_A_stop_error : BOOL;

	FilteratePump_P602_A_overload_Filter : ErrorFilter;
	FilteratePump_P602_A_incomplete_Filter : ErrorFilter;
	FilteratePump_P602_A_status_Filter : ErrorFilter;
	FilteratePump_P602_A_stop_Filter : ErrorFilter;


	FilteratePump_P602_B_remote_mode AT%I* : BOOL;
	FilteratePump_P602_B_overload AT%I* : BOOL;
	FilteratePump_P602_B_incomplete AT%I* : BOOL;
	FilteratePump_P602_B_status AT%I* : BOOL;

	FilteratePump_P602_B_command AT%Q* : BOOL;

	FilteratePump_P602_B_in : BOOL;
	FilteratePump_P602_B_overload_error : BOOL;
	FilteratePump_P602_B_incomplete_error : BOOL;
	FilteratePump_P602_B_status_error : BOOL;
	FilteratePump_P602_B_common_error : BOOL;
	FilteratePump_P602_B_stop_error : BOOL;

	FilteratePump_P602_B_overload_Filter : ErrorFilter;
	FilteratePump_P602_B_incomplete_Filter : ErrorFilter;
	FilteratePump_P602_B_status_Filter : ErrorFilter;
	FilteratePump_P602_B_stop_Filter : ErrorFilter;

	FilteratePump_P602_A :Equipment_Single;
	FilteratePump_P602_B :Equipment_Single;



	DrumThickener_D503_A_remote_mode AT%I* : BOOL;
	DrumThickener_D503_A_overload AT%I* : BOOL;
	DrumThickener_D503_A_incomplete AT%I* : BOOL;
	DrumThickener_D503_A_status AT%I* : BOOL;

	DrumThickener_D503_A_command AT%Q* : BOOL;

	DrumThickener_D503_A_in : BOOL;
	DrumThickener_D503_A_overload_error : BOOL;
	DrumThickener_D503_A_incomplete_error : BOOL;
	DrumThickener_D503_A_status_error : BOOL;
	DrumThickener_D503_A_common_error : BOOL;
	DrumThickener_D503_A_stop_error : BOOL;

	DrumThickener_D503_A_overload_Filter : ErrorFilter;
	DrumThickener_D503_A_incomplete_Filter : ErrorFilter;
	DrumThickener_D503_A_status_Filter : ErrorFilter;
	DrumThickener_D503_A_stop_Filter : ErrorFilter;


	DrumThickener_D503_B_remote_mode AT%I* : BOOL;
	DrumThickener_D503_B_overload AT%I* : BOOL;
	DrumThickener_D503_B_incomplete AT%I* : BOOL;
	DrumThickener_D503_B_status AT%I* : BOOL;

	DrumThickener_D503_B_command AT%Q* : BOOL;

	DrumThickener_D503_B_in : BOOL;
	DrumThickener_D503_B_overload_error : BOOL;
	DrumThickener_D503_B_incomplete_error : BOOL;
	DrumThickener_D503_B_status_error : BOOL;
	DrumThickener_D503_B_common_error : BOOL;
	DrumThickener_D503_B_stop_error : BOOL;

	DrumThickener_D503_B_overload_Filter : ErrorFilter;
	DrumThickener_D503_B_incomplete_Filter : ErrorFilter;
	DrumThickener_D503_B_status_Filter : ErrorFilter;
	DrumThickener_D503_B_stop_Filter : ErrorFilter;

	DrumThickener_D503_A :Equipment_Single;
	DrumThickener_D503_B :Equipment_Single;

	Floculator_M502_A_remote_mode AT%I* : BOOL;
	Floculator_M502_A_overload AT%I* : BOOL;
	Floculator_M502_A_incomplete AT%I* : BOOL;
	Floculator_M502_A_status AT%I* : BOOL;

	Floculator_M502_A_command AT%Q* : BOOL;

	Floculator_M502_A_in : BOOL;
	Floculator_M502_A_overload_error : BOOL;
	Floculator_M502_A_incomplete_error : BOOL;
	Floculator_M502_A_status_error : BOOL;
	Floculator_M502_A_common_error : BOOL;
	Floculator_M502_A_stop_error : BOOL;

	Floculator_M502_A_overload_Filter : ErrorFilter;
	Floculator_M502_A_incomplete_Filter : ErrorFilter;
	Floculator_M502_A_status_Filter : ErrorFilter;
	Floculator_M502_A_stop_Filter : ErrorFilter;


	Floculator_M502_B_remote_mode AT%I* : BOOL;
	Floculator_M502_B_overload AT%I* : BOOL;
	Floculator_M502_B_incomplete AT%I* : BOOL;
	Floculator_M502_B_status AT%I* : BOOL;

	Floculator_M502_B_command AT%Q* : BOOL;

	Floculator_M502_B_in : BOOL;
	Floculator_M502_B_overload_error : BOOL;
	Floculator_M502_B_incomplete_error : BOOL;
	Floculator_M502_B_status_error : BOOL;
	Floculator_M502_B_common_error : BOOL;
	Floculator_M502_B_stop_error : BOOL;

	Floculator_M502_B_overload_Filter : ErrorFilter;
	Floculator_M502_B_incomplete_Filter : ErrorFilter;
	Floculator_M502_B_status_Filter : ErrorFilter;
	Floculator_M502_B_stop_Filter : ErrorFilter;

	Floculator_M502_A : Equipment_Single;
	Floculator_M502_B :Equipment_Single;

	AirBlower_B501_A_remote_mode AT%I* : BOOL;
	AirBlower_B501_A_overload AT%I* : BOOL;
	AirBlower_B501_A_incomplete AT%I* : BOOL;
	AirBlower_B501_A_status AT%I* : BOOL;

	AirBlower_B501_A_command AT%Q* : BOOL;

	AirBlower_B501_A_in : BOOL;
	AirBlower_B501_A_overload_error : BOOL;
	AirBlower_B501_A_incomplete_error : BOOL;
	AirBlower_B501_A_status_error : BOOL;
	AirBlower_B501_A_common_error : BOOL;
	AirBlower_B501_A_stop_error : BOOL;

	AirBlower_B501_A_overload_Filter : ErrorFilter;
	AirBlower_B501_A_incomplete_Filter : ErrorFilter;
	AirBlower_B501_A_status_Filter : ErrorFilter;
	AirBlower_B501_A_stop_Filter : ErrorFilter;



	AirBlower_B501_B_remote_mode AT%I* : BOOL;
	AirBlower_B501_B_overload AT%I* : BOOL;
	AirBlower_B501_B_incomplete AT%I* : BOOL;
	AirBlower_B501_B_status AT%I* : BOOL;

	AirBlower_B501_B_command AT%Q* : BOOL;

	AirBlower_B501_B_in : BOOL;
	AirBlower_B501_B_overload_error : BOOL;
	AirBlower_B501_B_incomplete_error : BOOL;
	AirBlower_B501_B_status_error : BOOL;
	AirBlower_B501_B_common_error : BOOL;
	AirBlower_B501_B_stop_error : BOOL;

	AirBlower_B501_B_overload_Filter : ErrorFilter;
	AirBlower_B501_B_incomplete_Filter : ErrorFilter;
	AirBlower_B501_B_status_Filter : ErrorFilter;
	AirBlower_B501_B_stop_Filter : ErrorFilter;


	AirBlower_B501_C_remote_mode AT%I* : BOOL;
	AirBlower_B501_C_overload AT%I* : BOOL;
	AirBlower_B501_C_incomplete AT%I* : BOOL;
	AirBlower_B501_C_status AT%I* : BOOL;

	AirBlower_B501_C_command AT%Q* : BOOL;

	AirBlower_B501_C_in : BOOL;
	AirBlower_B501_C_overload_error : BOOL;
	AirBlower_B501_C_incomplete_error : BOOL;
	AirBlower_B501_C_status_error : BOOL;
	AirBlower_B501_C_common_error : BOOL;
	AirBlower_B501_C_stop_error : BOOL;

	AirBlower_B501_C_overload_Filter : ErrorFilter;
	AirBlower_B501_C_incomplete_Filter : ErrorFilter;
	AirBlower_B501_C_status_Filter : ErrorFilter;
	AirBlower_B501_C_stop_Filter : ErrorFilter;

	AirBlower_B501 :Equipment_Triple;

	BackwashWaterPump_P505_A_remote_mode AT%I* : BOOL;
	BackwashWaterPump_P505_A_overload AT%I* : BOOL;
	BackwashWaterPump_P505_A_incomplete AT%I* : BOOL;
	BackwashWaterPump_P505_A_status AT%I* : BOOL;

	BackwashWaterPump_P505_A_command AT%Q* : BOOL;

	BackwashWaterPump_P505_A_in : BOOL;
	BackwashWaterPump_P505_A_overload_error : BOOL;
	BackwashWaterPump_P505_A_incomplete_error : BOOL;
	BackwashWaterPump_P505_A_status_error : BOOL;
	BackwashWaterPump_P505_A_common_error : BOOL;
	BackwashWaterPump_P505_A_stop_error : BOOL;

	BackwashWaterPump_P505_A_overload_Filter : ErrorFilter;
	BackwashWaterPump_P505_A_incomplete_Filter : ErrorFilter;
	BackwashWaterPump_P505_A_status_Filter : ErrorFilter;
	BackwashWaterPump_P505_A_stop_Filter : ErrorFilter;



	BackwashWaterPump_P505_B_remote_mode AT%I* : BOOL;
	BackwashWaterPump_P505_B_overload AT%I* : BOOL;
	BackwashWaterPump_P505_B_incomplete AT%I* : BOOL;
	BackwashWaterPump_P505_B_status AT%I* : BOOL;

	BackwashWaterPump_P505_B_command AT%Q* : BOOL;

	BackwashWaterPump_P505_B_in : BOOL;
	BackwashWaterPump_P505_B_overload_error : BOOL;
	BackwashWaterPump_P505_B_incomplete_error : BOOL;
	BackwashWaterPump_P505_B_status_error : BOOL;
	BackwashWaterPump_P505_B_common_error : BOOL;
	BackwashWaterPump_P505_B_stop_error : BOOL;

	BackwashWaterPump_P505_B_overload_Filter : ErrorFilter;
	BackwashWaterPump_P505_B_incomplete_Filter : ErrorFilter;
	BackwashWaterPump_P505_B_status_Filter : ErrorFilter;
	BackwashWaterPump_P505_B_stop_Filter : ErrorFilter;



	BackwashWaterPump_P505_C_remote_mode AT%I* : BOOL;
	BackwashWaterPump_P505_C_overload AT%I* : BOOL;
	BackwashWaterPump_P505_C_incomplete AT%I* : BOOL;
	BackwashWaterPump_P505_C_status AT%I* : BOOL;

	BackwashWaterPump_P505_C_command AT%Q* : BOOL;

	BackwashWaterPump_P505_C_in : BOOL;
	BackwashWaterPump_P505_C_overload_error : BOOL;
	BackwashWaterPump_P505_C_incomplete_error : BOOL;
	BackwashWaterPump_P505_C_status_error : BOOL;
	BackwashWaterPump_P505_C_common_error : BOOL;
	BackwashWaterPump_P505_C_stop_error : BOOL;

	BackwashWaterPump_P505_C_overload_Filter : ErrorFilter;
	BackwashWaterPump_P505_C_incomplete_Filter : ErrorFilter;
	BackwashWaterPump_P505_C_status_Filter : ErrorFilter;
	BackwashWaterPump_P505_C_stop_Filter : ErrorFilter;

	BackwashWaterPump_P505 :Equipment_Triple;

END_VAR
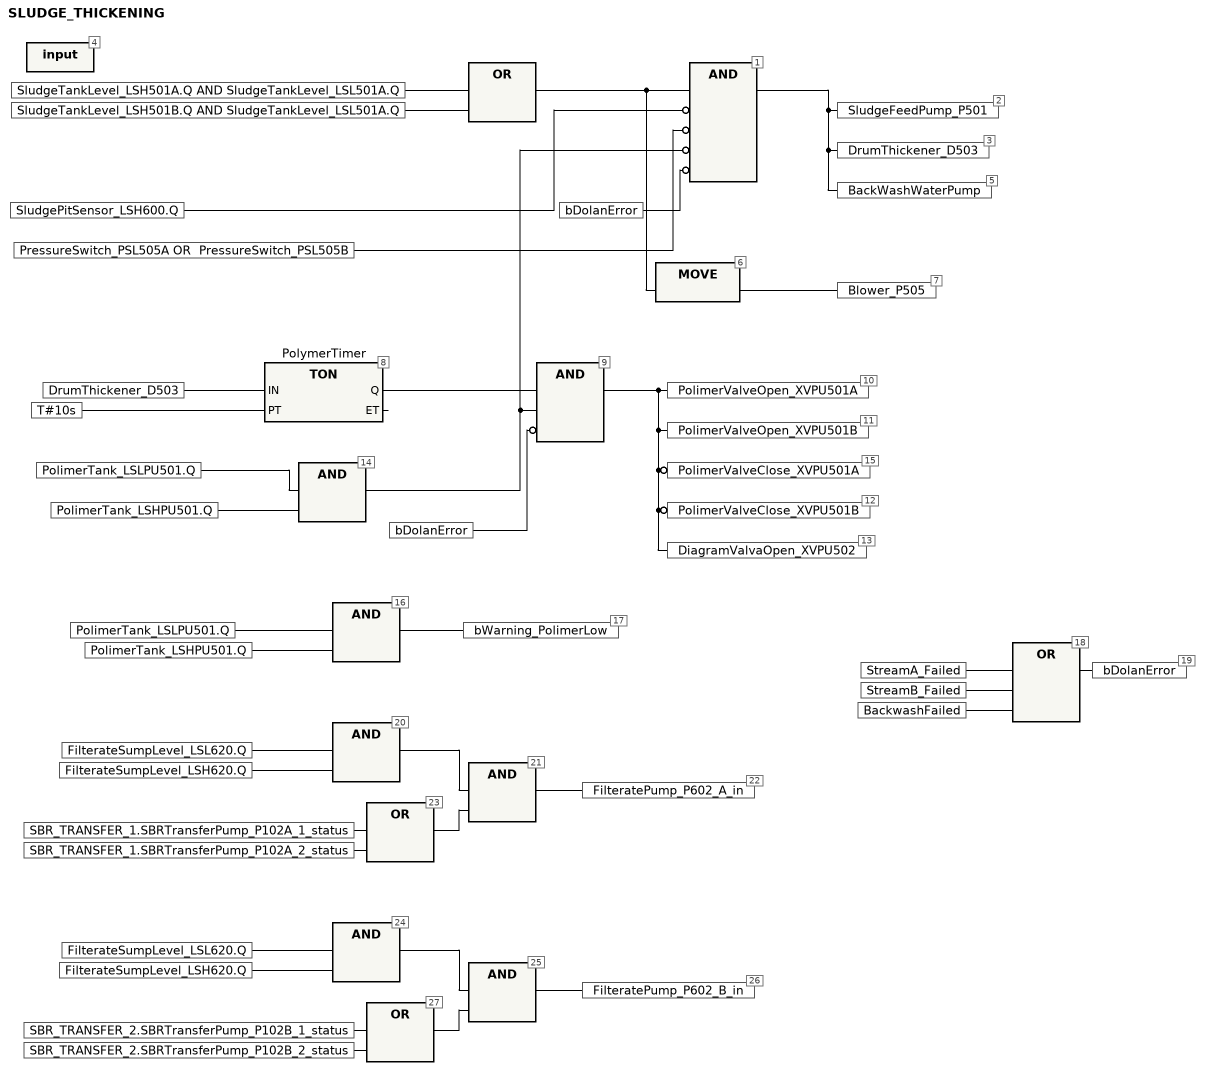
_CFC_ (* Continuous Function Chart, elements in execution order *)
#0 OR(SludgeTankLevel_LSH501A.Q AND SludgeTankLevel_LSL501A.Q, SludgeTankLevel_LSH501B.Q AND SludgeTankLevel_LSL501A.Q)
#1 AND(#0, NOT SludgePitSensor_LSH600.Q, NOT PressureSwitch_PSL505A OR PressureSwitch_PSL505B, NOT #14, NOT bDolanError)
#2 SludgeFeedPump_P501 <= #1
#3 DrumThickener_D503 <= #1
#4 input()
#5 BackWashWaterPump <= #1
#6 MOVE(#0)
#7 Blower_P505 <= #6
#8 PolymerTimer:TON(IN: DrumThickener_D503, PT: T#10s)
#9 AND(#8.Q, #14, NOT bDolanError)
#10 PolimerValveOpen_XVPU501A <= #9
#11 PolimerValveOpen_XVPU501B <= #9
#12 PolimerValveClose_XVPU501B <= NOT #9
#13 DiagramValvaOpen_XVPU502 <= #9
#14 AND(PolimerTank_LSLPU501.Q, PolimerTank_LSHPU501.Q)
#15 PolimerValveClose_XVPU501A <= NOT #9
#16 AND(PolimerTank_LSLPU501.Q, PolimerTank_LSHPU501.Q)
#17 bWarning_PolimerLow <= #16
#18 OR(StreamA_Failed, StreamB_Failed, BackwashFailed)
#19 bDolanError <= #18
#20 AND(FilterateSumpLevel_LSL620.Q, FilterateSumpLevel_LSH620.Q)
#21 AND(#20, #23)
#22 FilteratePump_P602_A_in <= #21
#23 OR(SBR_TRANSFER_1.SBRTransferPump_P102A_1_status, SBR_TRANSFER_1.SBRTransferPump_P102A_2_status)
#24 AND(FilterateSumpLevel_LSL620.Q, FilterateSumpLevel_LSH620.Q)
#25 AND(#24, #27)
#26 FilteratePump_P602_B_in <= #25
#27 OR(SBR_TRANSFER_2.SBRTransferPump_P102B_1_status, SBR_TRANSFER_2.SBRTransferPump_P102B_2_status)
_END_CFC_
END_PROGRAM
ACTION input:
	SludgeTankLevel_LSH501A();
	SludgeTankLevel_LSH501B();
	SludgeTankLevel_LSL501A();
	SludgeTankLevel_LSL501B();
	SludgePitSensor_LSH600();
	PolimerTank_LSLPU501();
	PolimerTank_LSHPU501();
	FilterateSumpLevel_LSL620();
	FilterateSumpLevel_LSH620();


FilteratePump_P602_A_overload_Filter(IN:=(FilteratePump_P602_A_overload AND FilteratePump_P602_A_in),PT:=T#2s,Q=>FilteratePump_P602_A_overload_error);
FilteratePump_P602_A_incomplete_Filter(IN:=(FilteratePump_P602_A_incomplete AND FilteratePump_P602_A_in),PT:=T#2s,Q=>FilteratePump_P602_A_incomplete_error);
FilteratePump_P602_A_status_Filter(IN:=(NOT FilteratePump_P602_A_status AND FilteratePump_P602_A_in),PT:=T#10s, Q=>FilteratePump_P602_A_status_error);
FilteratePump_P602_A_stop_Filter(IN:=( FilteratePump_P602_A_status AND NOT FilteratePump_P602_A_in),PT:=T#10s, Q=>FilteratePump_P602_A_stop_error);

FilteratePump_P602_A_common_error := FilteratePump_P602_A_overload_error OR FilteratePump_P602_A_incomplete_error OR FilteratePump_P602_A_status_error OR FilteratePump_P602_A_stop_error;



FilteratePump_P602_B_overload_Filter(IN:=(FilteratePump_P602_B_overload AND FilteratePump_P602_B_in),PT:=T#2s,Q=>FilteratePump_P602_B_overload_error);
FilteratePump_P602_B_incomplete_Filter(IN:=(FilteratePump_P602_B_incomplete AND FilteratePump_P602_B_in),PT:=T#2s,Q=>FilteratePump_P602_B_incomplete_error);
FilteratePump_P602_B_status_Filter(IN:=(NOT FilteratePump_P602_B_status AND FilteratePump_P602_B_in),PT:=T#10s, Q=>FilteratePump_P602_B_status_error);
FilteratePump_P602_B_stop_Filter(IN:=( FilteratePump_P602_B_status AND NOT FilteratePump_P602_B_in),PT:=T#10s, Q=>FilteratePump_P602_B_stop_error);

FilteratePump_P602_B_common_error := FilteratePump_P602_B_overload_error OR FilteratePump_P602_B_incomplete_error OR FilteratePump_P602_B_status_error OR FilteratePump_P602_B_stop_error;

FilteratePump_P602_A(
	ERROR1:=FilteratePump_P602_A_common_error ,
	remote1:=FilteratePump_P602_A_remote_mode ,
	IN1:=FilteratePump_P602_A_in ,
	Command1=> FilteratePump_P602_A_command);

FilteratePump_P602_B(
	ERROR1:=FilteratePump_P602_B_common_error ,
	remote1:=FilteratePump_P602_B_remote_mode ,
	IN1:=FilteratePump_P602_B_in ,
	Command1=> FilteratePump_P602_B_command);


DrumThickener_D503_A_overload_Filter(IN:=(DrumThickener_D503_A_overload AND DrumThickener_D503_A_in),PT:=T#2s,Q=>DrumThickener_D503_A_overload_error);
DrumThickener_D503_A_incomplete_Filter(IN:=(DrumThickener_D503_A_incomplete AND DrumThickener_D503_A_in),PT:=T#2s,Q=>DrumThickener_D503_A_incomplete_error);
DrumThickener_D503_A_status_Filter(IN:=(NOT DrumThickener_D503_A_status AND DrumThickener_D503_A_in),PT:=T#10s, Q=>DrumThickener_D503_A_status_error);
DrumThickener_D503_A_stop_Filter(IN:=( DrumThickener_D503_A_status AND NOT DrumThickener_D503_A_in),PT:=T#10s, Q=>DrumThickener_D503_A_stop_error);

DrumThickener_D503_A_common_error := DrumThickener_D503_A_overload_error OR DrumThickener_D503_A_incomplete_error OR DrumThickener_D503_A_status_error OR DrumThickener_D503_A_stop_error;


DrumThickener_D503_B_overload_Filter(IN:=(DrumThickener_D503_B_overload AND DrumThickener_D503_B_in),PT:=T#2s,Q=>DrumThickener_D503_B_overload_error);
DrumThickener_D503_B_incomplete_Filter(IN:=(DrumThickener_D503_B_incomplete AND DrumThickener_D503_B_in),PT:=T#2s,Q=>DrumThickener_D503_B_incomplete_error);
DrumThickener_D503_B_status_Filter(IN:=(NOT DrumThickener_D503_B_status AND DrumThickener_D503_B_in),PT:=T#10s, Q=>DrumThickener_D503_B_status_error);
DrumThickener_D503_B_stop_Filter(IN:=( DrumThickener_D503_B_status AND NOT DrumThickener_D503_B_in),PT:=T#10s, Q=>DrumThickener_D503_B_stop_error);

DrumThickener_D503_B_common_error := DrumThickener_D503_B_overload_error OR DrumThickener_D503_B_incomplete_error OR DrumThickener_D503_B_status_error OR DrumThickener_D503_B_stop_error;

DrumThickener_D503_A_in := DrumThickener_D503;
DrumThickener_D503_A(
	ERROR1:=DrumThickener_D503_A_common_error ,
	remote1:=DrumThickener_D503_A_remote_mode ,
	IN1:=DrumThickener_D503_A_in ,
	Command1=>DrumThickener_D503_A_command );

DrumThickener_D503_B_in := DrumThickener_D503;
DrumThickener_D503_B(
	ERROR1:=DrumThickener_D503_B_common_error ,
	remote1:=DrumThickener_D503_B_remote_mode ,
	IN1:=DrumThickener_D503_B_in ,
	Command1=>DrumThickener_D503_B_command );


bFloculator_M502A := DrumThickener_D503_A_command;
SolenoidValve_XV505A := DrumThickener_D503_A_command;

bFloculator_M502B := DrumThickener_D503_B_command;
SolenoidValve_XV505B := DrumThickener_D503_B_command;


Floculator_M502_A_overload_Filter(IN:=(Floculator_M502_A_overload AND Floculator_M502_A_in),PT:=T#2s,Q=>Floculator_M502_A_overload_error);
Floculator_M502_A_incomplete_Filter(IN:=(Floculator_M502_A_incomplete AND Floculator_M502_A_in),PT:=T#2s,Q=>Floculator_M502_A_incomplete_error);
Floculator_M502_A_status_Filter(IN:=(NOT Floculator_M502_A_status AND Floculator_M502_A_in),PT:=T#10s, Q=>Floculator_M502_A_status_error);
Floculator_M502_A_stop_Filter(IN:=( Floculator_M502_A_status AND NOT Floculator_M502_A_in),PT:=T#10s, Q=>Floculator_M502_A_stop_error);

Floculator_M502_A_common_error := Floculator_M502_A_overload_error OR Floculator_M502_A_incomplete_error OR Floculator_M502_A_status_error OR Floculator_M502_A_stop_error;



Floculator_M502_B_overload_Filter(IN:=(Floculator_M502_B_overload AND Floculator_M502_B_in),PT:=T#2s,Q=>Floculator_M502_B_overload_error);
Floculator_M502_B_incomplete_Filter(IN:=(Floculator_M502_B_incomplete AND Floculator_M502_B_in),PT:=T#2s,Q=>Floculator_M502_B_incomplete_error);
Floculator_M502_B_status_Filter(IN:=(NOT Floculator_M502_B_status AND Floculator_M502_B_in),PT:=T#10s, Q=>Floculator_M502_B_status_error);
Floculator_M502_B_stop_Filter(IN:=( Floculator_M502_B_status AND NOT Floculator_M502_B_in),PT:=T#10s, Q=>Floculator_M502_B_stop_error);

Floculator_M502_B_common_error := Floculator_M502_B_overload_error OR Floculator_M502_B_incomplete_error OR Floculator_M502_B_status_error OR Floculator_M502_B_stop_error;


Floculator_M502_A(
	ERROR1:=Floculator_M502_A_common_error ,
	remote1:= Floculator_M502_A_remote_mode,
	IN1:= Floculator_M502_A_in,
	Command1=>Floculator_M502_A_command);

Floculator_M502_B(
	ERROR1:=Floculator_M502_B_common_error ,
	remote1:= Floculator_M502_B_remote_mode,
	IN1:= Floculator_M502_B_in,
	Command1=>Floculator_M502_B_command);

StreamA_Failed := Floculator_M502_A_common_error AND DrumThickener_D503_A_common_error;
StreamB_Failed := Floculator_M502_B_common_error AND DrumThickener_D503_B_common_error;

AirBlower_B501_A_overload_Filter(IN:=(AirBlower_B501_A_overload AND AirBlower_B501_A_in),PT:=T#2s,Q=>AirBlower_B501_A_overload_error);
AirBlower_B501_A_incomplete_Filter(IN:=(AirBlower_B501_A_incomplete AND AirBlower_B501_A_in),PT:=T#2s,Q=>AirBlower_B501_A_incomplete_error);
AirBlower_B501_A_status_Filter(IN:=(NOT AirBlower_B501_A_status AND AirBlower_B501_A_in),PT:=T#10s, Q=>AirBlower_B501_A_status_error);
AirBlower_B501_A_stop_Filter(IN:=( AirBlower_B501_A_status AND NOT AirBlower_B501_A_in),PT:=T#10s, Q=>AirBlower_B501_A_stop_error);

AirBlower_B501_A_common_error := AirBlower_B501_A_overload_error OR AirBlower_B501_A_incomplete_error OR AirBlower_B501_A_status_error OR AirBlower_B501_A_stop_error;



AirBlower_B501_B_overload_Filter(IN:=(AirBlower_B501_B_overload AND AirBlower_B501_B_in),PT:=T#2s,Q=>AirBlower_B501_B_overload_error);
AirBlower_B501_B_incomplete_Filter(IN:=(AirBlower_B501_B_incomplete AND AirBlower_B501_B_in),PT:=T#2s,Q=>AirBlower_B501_B_incomplete_error);
AirBlower_B501_B_status_Filter(IN:=(NOT AirBlower_B501_B_status AND AirBlower_B501_B_in),PT:=T#10s, Q=>AirBlower_B501_B_status_error);
AirBlower_B501_B_stop_Filter(IN:=( AirBlower_B501_B_status AND NOT AirBlower_B501_B_in),PT:=T#10s, Q=>AirBlower_B501_B_stop_error);

AirBlower_B501_B_common_error := AirBlower_B501_B_overload_error OR AirBlower_B501_B_incomplete_error OR AirBlower_B501_B_status_error OR AirBlower_B501_B_stop_error;



AirBlower_B501_C_overload_Filter(IN:=(AirBlower_B501_C_overload AND AirBlower_B501_C_in),PT:=T#2s,Q=>AirBlower_B501_C_overload_error);
AirBlower_B501_C_incomplete_Filter(IN:=(AirBlower_B501_C_incomplete AND AirBlower_B501_C_in),PT:=T#2s,Q=>AirBlower_B501_C_incomplete_error);
AirBlower_B501_C_status_Filter(IN:=(NOT AirBlower_B501_C_status AND AirBlower_B501_C_in),PT:=T#10s, Q=>AirBlower_B501_C_status_error);
AirBlower_B501_C_stop_Filter(IN:=( AirBlower_B501_C_status AND NOT AirBlower_B501_C_in),PT:=T#10s, Q=>AirBlower_B501_C_stop_error);

AirBlower_B501_C_common_error := AirBlower_B501_C_overload_error OR AirBlower_B501_C_incomplete_error OR AirBlower_B501_C_status_error OR AirBlower_B501_C_stop_error;

AirBlower_B501_A_in := Blower_P505;
AirBlower_B501_B_in := Blower_P505;

AirBlower_B501(
	ERROR1:=AirBlower_B501_A_common_error ,
	ERROR2:=AirBlower_B501_C_common_error ,
	ERROR3:=AirBlower_B501_B_common_error ,
	remote1:=AirBlower_B501_A_remote_mode ,
	remote2:=AirBlower_B501_C_remote_mode,
	remote3:= AirBlower_B501_B_remote_mode,
	IN1:=AirBlower_B501_A_in ,
	IN2:=AirBlower_B501_C_in ,
	IN3:=AirBlower_B501_B_in ,
	Command1=>AirBlower_B501_A_command ,
	Command2=>AirBlower_B501_C_command ,
	Command3=>AirBlower_B501_B_command );

BlowerValve_XV501A := AirBlower_B501_A_common_error;
BlowerValve_XV501B := AirBlower_B501_C_common_error;

BackwashWaterPump_P505_A_overload_Filter(IN:=(BackwashWaterPump_P505_A_overload AND BackwashWaterPump_P505_A_in),PT:=T#2s,Q=>BackwashWaterPump_P505_A_overload_error);
BackwashWaterPump_P505_A_incomplete_Filter(IN:=(BackwashWaterPump_P505_A_incomplete AND BackwashWaterPump_P505_A_in),PT:=T#2s,Q=>BackwashWaterPump_P505_A_incomplete_error);
BackwashWaterPump_P505_A_status_Filter(IN:=(NOT BackwashWaterPump_P505_A_status AND BackwashWaterPump_P505_A_in),PT:=T#10s, Q=>BackwashWaterPump_P505_A_status_error);
BackwashWaterPump_P505_A_stop_Filter(IN:=( BackwashWaterPump_P505_A_status AND NOT BackwashWaterPump_P505_A_in),PT:=T#10s, Q=>BackwashWaterPump_P505_A_stop_error);

BackwashWaterPump_P505_A_common_error := BackwashWaterPump_P505_A_overload_error OR BackwashWaterPump_P505_A_incomplete_error OR BackwashWaterPump_P505_A_status_error OR BackwashWaterPump_P505_A_stop_error;


BackwashWaterPump_P505_B_overload_Filter(IN:=(BackwashWaterPump_P505_B_overload AND BackwashWaterPump_P505_B_in),PT:=T#2s,Q=>BackwashWaterPump_P505_B_overload_error);
BackwashWaterPump_P505_B_incomplete_Filter(IN:=(BackwashWaterPump_P505_B_incomplete AND BackwashWaterPump_P505_B_in),PT:=T#2s,Q=>BackwashWaterPump_P505_B_incomplete_error);
BackwashWaterPump_P505_B_status_Filter(IN:=(NOT BackwashWaterPump_P505_B_status AND BackwashWaterPump_P505_B_in),PT:=T#10s, Q=>BackwashWaterPump_P505_B_status_error);
BackwashWaterPump_P505_B_stop_Filter(IN:=( BackwashWaterPump_P505_B_status AND NOT BackwashWaterPump_P505_B_in),PT:=T#10s, Q=>BackwashWaterPump_P505_B_stop_error);

BackwashWaterPump_P505_B_common_error := BackwashWaterPump_P505_B_overload_error OR BackwashWaterPump_P505_B_incomplete_error OR BackwashWaterPump_P505_B_status_error OR BackwashWaterPump_P505_B_stop_error;


BackwashWaterPump_P505_C_overload_Filter(IN:=(BackwashWaterPump_P505_C_overload AND BackwashWaterPump_P505_C_in),PT:=T#2s,Q=>BackwashWaterPump_P505_C_overload_error);
BackwashWaterPump_P505_C_incomplete_Filter(IN:=(BackwashWaterPump_P505_C_incomplete AND BackwashWaterPump_P505_C_in),PT:=T#2s,Q=>BackwashWaterPump_P505_C_incomplete_error);
BackwashWaterPump_P505_C_status_Filter(IN:=(NOT BackwashWaterPump_P505_C_status AND BackwashWaterPump_P505_C_in),PT:=T#10s, Q=>BackwashWaterPump_P505_C_status_error);
BackwashWaterPump_P505_C_stop_Filter(IN:=( BackwashWaterPump_P505_C_status AND NOT BackwashWaterPump_P505_C_in),PT:=T#10s, Q=>BackwashWaterPump_P505_C_stop_error);

BackwashWaterPump_P505_C_common_error := BackwashWaterPump_P505_C_overload_error OR BackwashWaterPump_P505_C_incomplete_error OR BackwashWaterPump_P505_C_status_error OR BackwashWaterPump_P505_C_stop_error;

BackwashWaterPump_P505_A_in := BackWashWaterPump;
BackwashWaterPump_P505_B_in := BackWashWaterPump;

BackWashWaterPump_P505(
	ERROR1:=BackwashWaterPump_P505_A_common_error ,
	ERROR2:=BackwashWaterPump_P505_B_common_error ,
	ERROR3:=BackwashWaterPump_P505_C_common_error ,
	remote1:= BackwashWaterPump_P505_A_remote_mode,
	remote2:=BackwashWaterPump_P505_B_remote_mode ,
	remote3:=BackwashWaterPump_P505_C_remote_mode ,
	IN1:=BackwashWaterPump_P505_A_in ,
	IN2:=BackwashWaterPump_P505_B_in ,
	IN3:=BackwashWaterPump_P505_C_in ,
	Command1=>BackwashWaterPump_P505_A_command ,
	Command2=>BackwashWaterPump_P505_B_command ,
	Command3=>BackwashWaterPump_P505_C_command );

BackwashFailed :=( BackwashWaterPump_P505_A_common_error OR BackwashWaterPump_P505_B_common_error) AND BackwashWaterPump_P505_C_common_error;
END_ACTION

(* POU module/Equipment_Single, ST *)
FUNCTION_BLOCK Equipment_Single
VAR_INPUT
	ERROR1 : BOOL;
	remote1 : BOOL;
END_VAR
VAR_OUTPUT
	Command1 : BOOL;
END_VAR
VAR_IN_OUT
	IN1 : BOOL;
END_VAR
Command1 := IN1 AND remote1;
END_FUNCTION_BLOCK

(* POU module/Equipment_Triple, ST *)
FUNCTION_BLOCK Equipment_Triple
VAR_INPUT
	ERROR1 : BOOL;
	ERROR2 : BOOL;
	ERROR3 : BOOL;
	remote1 : BOOL;
	remote2 : BOOL;
	remote3 : BOOL;
END_VAR
VAR_OUTPUT
	Command1 : BOOL;
	Command2 : BOOL;
	Command3 : BOOL;
END_VAR
VAR_IN_OUT
	IN1 : BOOL;
	IN2 : BOOL;
	IN3 : BOOL;
END_VAR
Command1 := IN1 AND remote1;
Command2 := IN2 AND remote2;
Command3 := IN3 AND remote3;
IN3 := ERROR1 OR ERROR2 AND (IN1 OR IN2);
END_FUNCTION_BLOCK

(* POU SBR_TRANSFER_2, CFC *)
PROGRAM SBR_TRANSFER_2
VAR
	LSL103B : inBlock;
	LSS103B : inBlock;
	LSH103B : inBlock;
	LSD103B : inBlock;


	bWarningSBRDry: BOOL;
	bCriticalSBRDry: BOOL;
	bCriticalSBRHi: BOOL;



	SBRTransferPump_P102B_1_remote_mode AT%I* : BOOL;
	SBRTransferPump_P102B_1_overload AT%I* : BOOL;
	SBRTransferPump_P102B_1_incomplete AT%I* : BOOL;
	SBRTransferPump_P102B_1_status AT%I* : BOOL;

	SBRTransferPump_P102B_1_command AT%Q* : BOOL;

	SBRTransferPump_P102B_1_in : BOOL;
	SBRTransferPump_P102B_1_overload_error : BOOL;
	SBRTransferPump_P102B_1_incomplete_error : BOOL;
	SBRTransferPump_P102B_1_status_error : BOOL;
	SBRTransferPump_P102B_1_common_error : BOOL;
	SBRTransferPump_P102B_1_stop_error : BOOL;

	SBRTransferPump_P102B_1_overload_Filter : ErrorFilter;
	SBRTransferPump_P102B_1_incomplete_Filter : ErrorFilter;
	SBRTransferPump_P102B_1_status_Filter : ErrorFilter;
	SBRTransferPump_P102B_1_stop_Filter : ErrorFilter;



	SBRTransferPump_P102B_2_remote_mode AT%I* : BOOL;
	SBRTransferPump_P102B_2_overload AT%I* : BOOL;
	SBRTransferPump_P102B_2_incomplete AT%I* : BOOL;
	SBRTransferPump_P102B_2_status AT%I* : BOOL;

	SBRTransferPump_P102B_2_command AT%Q* : BOOL;

	SBRTransferPump_P102B_2_in : BOOL;
	SBRTransferPump_P102B_2_overload_error : BOOL;
	SBRTransferPump_P102B_2_incomplete_error : BOOL;
	SBRTransferPump_P102B_2_status_error : BOOL;
	SBRTransferPump_P102B_2_common_error : BOOL;
	SBRTransferPump_P102B_2_stop_error : BOOL;

	SBRTransferPump_P102B_2_overload_Filter : ErrorFilter;
	SBRTransferPump_P102B_2_incomplete_Filter : ErrorFilter;
	SBRTransferPump_P102B_2_status_Filter : ErrorFilter;
	SBRTransferPump_P102B_2_stop_Filter : ErrorFilter;
	SBRTransferPump_P102B_CriticalStartingError: BOOL;
	SBRTransferPump_P102B: Equipment_Dual;
END_VAR
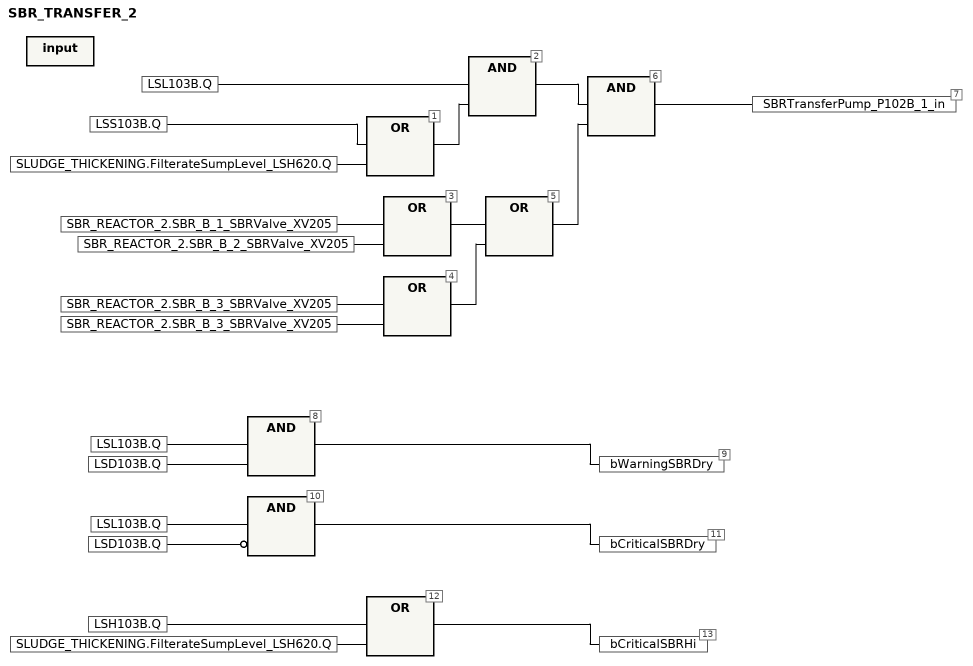
_CFC_ (* Continuous Function Chart, elements in execution order *)
#0 input()
#1 OR(LSS103B.Q, SLUDGE_THICKENING.FilterateSumpLevel_LSH620.Q)
#2 AND(LSL103B.Q, #1)
#3 OR(SBR_REACTOR_2.SBR_B_1_SBRValve_XV205, SBR_REACTOR_2.SBR_B_2_SBRValve_XV205)
#4 OR(SBR_REACTOR_2.SBR_B_3_SBRValve_XV205, SBR_REACTOR_2.SBR_B_3_SBRValve_XV205)
#5 OR(#3, #4)
#6 AND(#2, #5)
#7 SBRTransferPump_P102B_1_in <= #6
#8 AND(LSL103B.Q, LSD103B.Q)
#9 bWarningSBRDry <= #8
#10 AND(LSL103B.Q, NOT LSD103B.Q)
#11 bCriticalSBRDry <= #10
#12 OR(LSH103B.Q, SLUDGE_THICKENING.FilterateSumpLevel_LSH620.Q)
#13 bCriticalSBRHi <= #12
_END_CFC_
(* the same logic as Structured Text *)
input();
SBRTransferPump_P102B_1_in := (LSL103B.Q AND (LSS103B.Q OR SLUDGE_THICKENING.FilterateSumpLevel_LSH620.Q)) AND ((SBR_REACTOR_2.SBR_B_1_SBRValve_XV205 OR SBR_REACTOR_2.SBR_B_2_SBRValve_XV205) OR (SBR_REACTOR_2.SBR_B_3_SBRValve_XV205 OR SBR_REACTOR_2.SBR_B_3_SBRValve_XV205));
bWarningSBRDry := LSL103B.Q AND LSD103B.Q;
bCriticalSBRDry := LSL103B.Q AND NOT LSD103B.Q;
bCriticalSBRHi := LSH103B.Q OR SLUDGE_THICKENING.FilterateSumpLevel_LSH620.Q;
END_PROGRAM
ACTION Input:
LSD103B( );
LSH103B();
LSL103B( );
LSS103B( );

SBRTransferPump_P102B_1_overload_Filter(IN:=(SBRTransferPump_P102B_1_overload AND SBRTransferPump_P102B_1_in),PT:=T#2s,Q=>SBRTransferPump_P102B_1_overload_error);
SBRTransferPump_P102B_1_incomplete_Filter(IN:=(SBRTransferPump_P102B_1_incomplete AND SBRTransferPump_P102B_1_in),PT:=T#2s,Q=>SBRTransferPump_P102B_1_incomplete_error);
SBRTransferPump_P102B_1_status_Filter(IN:=(NOT SBRTransferPump_P102B_1_status AND SBRTransferPump_P102B_1_in),PT:=T#10s, Q=>SBRTransferPump_P102B_1_status_error);
SBRTransferPump_P102B_1_stop_Filter(IN:=( SBRTransferPump_P102B_1_status AND NOT SBRTransferPump_P102B_1_in),PT:=T#10s, Q=>SBRTransferPump_P102B_1_stop_error);

SBRTransferPump_P102B_1_common_error := SBRTransferPump_P102B_1_overload_error OR SBRTransferPump_P102B_1_incomplete_error OR SBRTransferPump_P102B_1_status_error OR SBRTransferPump_P102B_1_stop_error;


SBRTransferPump_P102B_2_overload_Filter(IN:=(SBRTransferPump_P102B_2_overload AND SBRTransferPump_P102B_2_in),PT:=T#2s,Q=>SBRTransferPump_P102B_2_overload_error);
SBRTransferPump_P102B_2_incomplete_Filter(IN:=(SBRTransferPump_P102B_2_incomplete AND SBRTransferPump_P102B_2_in),PT:=T#2s,Q=>SBRTransferPump_P102B_2_incomplete_error);
SBRTransferPump_P102B_2_status_Filter(IN:=(NOT SBRTransferPump_P102B_2_status AND SBRTransferPump_P102B_2_in),PT:=T#10s, Q=>SBRTransferPump_P102B_2_status_error);
SBRTransferPump_P102B_2_stop_Filter(IN:=( SBRTransferPump_P102B_2_status AND NOT SBRTransferPump_P102B_2_in),PT:=T#10s, Q=>SBRTransferPump_P102B_2_stop_error);

SBRTransferPump_P102B_2_common_error := SBRTransferPump_P102B_2_overload_error OR SBRTransferPump_P102B_2_incomplete_error OR SBRTransferPump_P102B_2_status_error OR SBRTransferPump_P102B_2_stop_error;

SBRTransferPump_P102B_CriticalStartingError := SBRTransferPump_P102B_1_common_error AND SBRTransferPump_P102B_2_common_error;

SBRTransferPump_P102B(
	ERROR1:=SBRTransferPump_P102B_1_common_error ,
	ERROR2:=SBRTransferPump_P102B_2_common_error ,
	remote1:=SBRTransferPump_P102B_1_remote_mode ,
	remote2:=SBRTransferPump_P102B_2_remote_mode ,
	IN1:= SBRTransferPump_P102B_1_in,
	IN2:=SBRTransferPump_P102B_2_in ,
	Command1=>SBRTransferPump_P102B_1_command ,
	Command2=>SBRTransferPump_P102B_2_command );
END_ACTION

(* POU SBR_REACTOR_2, CFC *)
PROGRAM SBR_REACTOR_2
VAR

	bDeSludge: BOOL;
	bBlower: BOOL;
	TimerStartBlower1: TON;
	TimerStartBlower2: TON;
	TimerStartBlower3: TON;
	tBlower1: fb_timer_on_off;
	tBlower2: fb_timer_on_off;
	tBlower3: fb_timer_on_off;



	SBR_B_1_SBRLevelSensor_LSH200 AT%I* : BOOL;
	SBR_B_1_DOSensor_DO201 AT%I* : INT;
	SBR_B_1_DecanterLevelSensorLow_Rx AT%I* : BOOL;
	SBR_B_1_DecanterLevelSensorHi_Rx AT%I* : BOOL;

	SBR_B_1_FowardDecant_XV26 AT%Q* : BOOL;
	SBR_B_1_ReverseDecant_XV26 AT%Q* : BOOL;
	SBR_B_1_BlowerValve_XV201 AT%Q* : BOOL;
	SBR_B_1_DeSludgeValve_XV241 AT%Q* : BOOL;
	SBR_B_1_SBRValve_XV205 AT%Q* : BOOL;
	SBR_B_1_SBRMixer_XV205  : BOOL;

	SBR_B_1_bEnable_SW : BOOL;
	SBR_B_1_Blower_B201 : BOOL;
	SBR_B_1_DesludgePump_P201 : BOOL;
	SBR_B_1_filling : BOOL;
	SBR_B_1_aeration : BOOL;
	SBR_B_1_settling : BOOL;
	SBR_B_1_decanting : BOOL;
	SBR_B_1_desludging : BOOL;
	SBR_B_1_SBRMixer_M200 : BOOL;
	SBR_B_1_warning_DONotInRange : BOOL;

	SBR_B_2_SBRLevelSensor_LSH200 AT%I* : BOOL;
	SBR_B_2_DOSensor_DO201 AT%I* : INT;
	SBR_B_2_DecanterLevelSensorLow_Rx AT%I* : BOOL;
	SBR_B_2_DecanterLevelSensorHi_Rx AT%I* : BOOL;

	SBR_B_2_FowardDecant_XV26 AT%Q* : BOOL;
	SBR_B_2_ReverseDecant_XV26 AT%Q* : BOOL;
	SBR_B_2_BlowerValve_XV201 AT%Q* : BOOL;
	SBR_B_2_DeSludgeValve_XV241 AT%Q* : BOOL;
	SBR_B_2_SBRValve_XV205 AT%Q* : BOOL;
	SBR_B_2_SBRMixer_XV205  : BOOL;

	SBR_B_2_bEnable_SW : BOOL;
	SBR_B_2_Blower_B201 : BOOL;
	SBR_B_2_DesludgePump_P201 : BOOL;
	SBR_B_2_filling : BOOL;
	SBR_B_2_aeration : BOOL;
	SBR_B_2_settling : BOOL;
	SBR_B_2_decanting : BOOL;
	SBR_B_2_desludging : BOOL;
	SBR_B_2_SBRMixer_M200 : BOOL;
	SBR_B_2_warning_DONotInRange : BOOL;

	SBR_B_3_SBRLevelSensor_LSH200 AT%I* : BOOL;
	SBR_B_3_DOSensor_DO201 AT%I* : INT;
	SBR_B_3_DecanterLevelSensorLow_Rx AT%I* : BOOL;
	SBR_B_3_DecanterLevelSensorHi_Rx AT%I* : BOOL;

	SBR_B_3_FowardDecant_XV26 AT%Q* : BOOL;
	SBR_B_3_ReverseDecant_XV26 AT%Q* : BOOL;
	SBR_B_3_BlowerValve_XV201 AT%Q* : BOOL;
	SBR_B_3_DeSludgeValve_XV241 AT%Q* : BOOL;
	SBR_B_3_SBRValve_XV205 AT%Q* : BOOL;
	SBR_B_3_SBRMixer_XV205  : BOOL;

	SBR_B_3_bEnable_SW : BOOL;
	SBR_B_3_Blower_B201 : BOOL;
	SBR_B_3_DesludgePump_P201 : BOOL;
	SBR_B_3_filling : BOOL;
	SBR_B_3_aeration : BOOL;
	SBR_B_3_settling : BOOL;
	SBR_B_3_decanting : BOOL;
	SBR_B_3_desludging : BOOL;
	SBR_B_3_SBRMixer_M200 : BOOL;
	SBR_B_3_warning_DONotInRange : BOOL;

	SBR_B_4_SBRLevelSensor_LSH200 AT%I* : BOOL;
	SBR_B_4_DOSensor_DO201 AT%I* : INT;
	SBR_B_4_DecanterLevelSensorLow_Rx AT%I* : BOOL;
	SBR_B_4_DecanterLevelSensorHi_Rx AT%I* : BOOL;

	SBR_B_4_FowardDecant_XV26 AT%Q* : BOOL;
	SBR_B_4_ReverseDecant_XV26 AT%Q* : BOOL;
	SBR_B_4_BlowerValve_XV201 AT%Q* : BOOL;
	SBR_B_4_DeSludgeValve_XV241 AT%Q* : BOOL;
	SBR_B_4_SBRValve_XV205 AT%Q* : BOOL;
	SBR_B_4_SBRMixer_XV205 : BOOL;

	SBR_B_4_bEnable_SW : BOOL;
	SBR_B_4_Blower_B201 : BOOL;
	SBR_B_4_DesludgePump_P201 : BOOL;
	SBR_B_4_filling : BOOL;
	SBR_B_4_aeration : BOOL;
	SBR_B_4_settling : BOOL;
	SBR_B_4_decanting : BOOL;
	SBR_B_4_desludging : BOOL;
	SBR_B_4_SBRMixer_M200 : BOOL;
	SBR_B_4_warning_DONotInRange : BOOL;


	SludeTankSensorLevelHi_LSL510B: inBlock;
	SBRReactor_1: SBRReactor;
	SBRReactor_2: SBRReactor;
	SBRReactor_3: SBRReactor;
	SBRReactor_4: SBRReactor;

	SBRMixer_M200B1_A_remote_mode AT%I* : BOOL;
	SBRMixer_M200B1_A_overload AT%I* : BOOL;
	SBRMixer_M200B1_A_incomplete AT%I* : BOOL;
	SBRMixer_M200B1_A_status AT%I* : BOOL;

	SBRMixer_M200B1_A_command AT%Q* : BOOL;

	SBRMixer_M200B1_A_in : BOOL;
	SBRMixer_M200B1_A_overload_error : BOOL;
	SBRMixer_M200B1_A_incomplete_error : BOOL;
	SBRMixer_M200B1_A_status_error : BOOL;
	SBRMixer_M200B1_A_common_error : BOOL;
	SBRMixer_M200B1_A_stop_error : BOOL;

	SBRMixer_M200B1_A_overload_Filter : ErrorFilter;
	SBRMixer_M200B1_A_incomplete_Filter : ErrorFilter;
	SBRMixer_M200B1_A_status_Filter : ErrorFilter;
	SBRMixer_M200B1_A_stop_Filter : ErrorFilter;

	SBRMixer_M200B1_B_remote_mode AT%I* : BOOL;
	SBRMixer_M200B1_B_overload AT%I* : BOOL;
	SBRMixer_M200B1_B_incomplete AT%I* : BOOL;
	SBRMixer_M200B1_B_status AT%I* : BOOL;

	SBRMixer_M200B1_B_command AT%Q* : BOOL;

	SBRMixer_M200B1_B_in : BOOL;
	SBRMixer_M200B1_B_overload_error : BOOL;
	SBRMixer_M200B1_B_incomplete_error : BOOL;
	SBRMixer_M200B1_B_status_error : BOOL;
	SBRMixer_M200B1_B_common_error : BOOL;
	SBRMixer_M200B1_B_stop_error : BOOL;

	SBRMixer_M200B1_B_overload_Filter : ErrorFilter;
	SBRMixer_M200B1_B_incomplete_Filter : ErrorFilter;
	SBRMixer_M200B1_B_status_Filter : ErrorFilter;
	SBRMixer_M200B1_B_stop_Filter : ErrorFilter;


	SBRMixer_M200B1_C_remote_mode AT%I* : BOOL;
	SBRMixer_M200B1_C_overload AT%I* : BOOL;
	SBRMixer_M200B1_C_incomplete AT%I* : BOOL;
	SBRMixer_M200B1_C_status AT%I* : BOOL;

	SBRMixer_M200B1_C_command AT%Q* : BOOL;

	SBRMixer_M200B1_C_in : BOOL;
	SBRMixer_M200B1_C_overload_error : BOOL;
	SBRMixer_M200B1_C_incomplete_error : BOOL;
	SBRMixer_M200B1_C_status_error : BOOL;
	SBRMixer_M200B1_C_common_error : BOOL;
	SBRMixer_M200B1_C_stop_error : BOOL;

	SBRMixer_M200B1_C_overload_Filter : ErrorFilter;
	SBRMixer_M200B1_C_incomplete_Filter : ErrorFilter;
	SBRMixer_M200B1_C_status_Filter : ErrorFilter;
	SBRMixer_M200B1_C_stop_Filter : ErrorFilter;



	SBRMixer_M200B2_A_remote_mode AT%I* : BOOL;
	SBRMixer_M200B2_A_overload AT%I* : BOOL;
	SBRMixer_M200B2_A_incomplete AT%I* : BOOL;
	SBRMixer_M200B2_A_status AT%I* : BOOL;

	SBRMixer_M200B2_A_command AT%Q* : BOOL;

	SBRMixer_M200B2_A_in : BOOL;
	SBRMixer_M200B2_A_overload_error : BOOL;
	SBRMixer_M200B2_A_incomplete_error : BOOL;
	SBRMixer_M200B2_A_status_error : BOOL;
	SBRMixer_M200B2_A_common_error : BOOL;
	SBRMixer_M200B2_A_stop_error : BOOL;

	SBRMixer_M200B2_A_overload_Filter : ErrorFilter;
	SBRMixer_M200B2_A_incomplete_Filter : ErrorFilter;
	SBRMixer_M200B2_A_status_Filter : ErrorFilter;
	SBRMixer_M200B2_A_stop_Filter : ErrorFilter;

	SBRMixer_M200B2_B_remote_mode AT%I* : BOOL;
	SBRMixer_M200B2_B_overload AT%I* : BOOL;
	SBRMixer_M200B2_B_incomplete AT%I* : BOOL;
	SBRMixer_M200B2_B_status AT%I* : BOOL;

	SBRMixer_M200B2_B_command AT%Q* : BOOL;

	SBRMixer_M200B2_B_in : BOOL;
	SBRMixer_M200B2_B_overload_error : BOOL;
	SBRMixer_M200B2_B_incomplete_error : BOOL;
	SBRMixer_M200B2_B_status_error : BOOL;
	SBRMixer_M200B2_B_common_error : BOOL;
	SBRMixer_M200B2_B_stop_error : BOOL;

	SBRMixer_M200B2_B_overload_Filter : ErrorFilter;
	SBRMixer_M200B2_B_incomplete_Filter : ErrorFilter;
	SBRMixer_M200B2_B_status_Filter : ErrorFilter;
	SBRMixer_M200B2_B_stop_Filter : ErrorFilter;


	SBRMixer_M200B2_C_remote_mode AT%I* : BOOL;
	SBRMixer_M200B2_C_overload AT%I* : BOOL;
	SBRMixer_M200B2_C_incomplete AT%I* : BOOL;
	SBRMixer_M200B2_C_status AT%I* : BOOL;

	SBRMixer_M200B2_C_command AT%Q* : BOOL;

	SBRMixer_M200B2_C_in : BOOL;
	SBRMixer_M200B2_C_overload_error : BOOL;
	SBRMixer_M200B2_C_incomplete_error : BOOL;
	SBRMixer_M200B2_C_status_error : BOOL;
	SBRMixer_M200B2_C_common_error : BOOL;
	SBRMixer_M200B2_C_stop_error : BOOL;

	SBRMixer_M200B2_C_overload_Filter : ErrorFilter;
	SBRMixer_M200B2_C_incomplete_Filter : ErrorFilter;
	SBRMixer_M200B2_C_status_Filter : ErrorFilter;
	SBRMixer_M200B2_C_stop_Filter : ErrorFilter;



	SBRMixer_M200B3_A_remote_mode AT%I* : BOOL;
	SBRMixer_M200B3_A_overload AT%I* : BOOL;
	SBRMixer_M200B3_A_incomplete AT%I* : BOOL;
	SBRMixer_M200B3_A_status AT%I* : BOOL;

	SBRMixer_M200B3_A_command AT%Q* : BOOL;

	SBRMixer_M200B3_A_in : BOOL;
	SBRMixer_M200B3_A_overload_error : BOOL;
	SBRMixer_M200B3_A_incomplete_error : BOOL;
	SBRMixer_M200B3_A_status_error : BOOL;
	SBRMixer_M200B3_A_common_error : BOOL;
	SBRMixer_M200B3_A_stop_error : BOOL;

	SBRMixer_M200B3_A_overload_Filter : ErrorFilter;
	SBRMixer_M200B3_A_incomplete_Filter : ErrorFilter;
	SBRMixer_M200B3_A_status_Filter : ErrorFilter;
	SBRMixer_M200B3_A_stop_Filter : ErrorFilter;

	SBRMixer_M200B3_B_remote_mode AT%I* : BOOL;
	SBRMixer_M200B3_B_overload AT%I* : BOOL;
	SBRMixer_M200B3_B_incomplete AT%I* : BOOL;
	SBRMixer_M200B3_B_status AT%I* : BOOL;

	SBRMixer_M200B3_B_command AT%Q* : BOOL;

	SBRMixer_M200B3_B_in : BOOL;
	SBRMixer_M200B3_B_overload_error : BOOL;
	SBRMixer_M200B3_B_incomplete_error : BOOL;
	SBRMixer_M200B3_B_status_error : BOOL;
	SBRMixer_M200B3_B_common_error : BOOL;
	SBRMixer_M200B3_B_stop_error : BOOL;

	SBRMixer_M200B3_B_overload_Filter : ErrorFilter;
	SBRMixer_M200B3_B_incomplete_Filter : ErrorFilter;
	SBRMixer_M200B3_B_status_Filter : ErrorFilter;
	SBRMixer_M200B3_B_stop_Filter : ErrorFilter;


	SBRMixer_M200B3_C_remote_mode AT%I* : BOOL;
	SBRMixer_M200B3_C_overload AT%I* : BOOL;
	SBRMixer_M200B3_C_incomplete AT%I* : BOOL;
	SBRMixer_M200B3_C_status AT%I* : BOOL;

	SBRMixer_M200B3_C_command AT%Q* : BOOL;

	SBRMixer_M200B3_C_in : BOOL;
	SBRMixer_M200B3_C_overload_error : BOOL;
	SBRMixer_M200B3_C_incomplete_error : BOOL;
	SBRMixer_M200B3_C_status_error : BOOL;
	SBRMixer_M200B3_C_common_error : BOOL;
	SBRMixer_M200B3_C_stop_error : BOOL;

	SBRMixer_M200B3_C_overload_Filter : ErrorFilter;
	SBRMixer_M200B3_C_incomplete_Filter : ErrorFilter;
	SBRMixer_M200B3_C_status_Filter : ErrorFilter;
	SBRMixer_M200B3_C_stop_Filter : ErrorFilter;

	DesludgePump_P201B_1_remote_mode AT%I* : BOOL;
	DesludgePump_P201B_1_overload AT%I* : BOOL;
	DesludgePump_P201B_1_incomplete AT%I* : BOOL;
	DesludgePump_P201B_1_status AT%I* : BOOL;

	DesludgePump_P201B_1_command AT%Q* : BOOL;

	DesludgePump_P201B_1_in : BOOL;
	DesludgePump_P201B_1_overload_error : BOOL;
	DesludgePump_P201B_1_incomplete_error : BOOL;
	DesludgePump_P201B_1_status_error : BOOL;
	DesludgePump_P201B_1_common_error : BOOL;
	DesludgePump_P201B_1_stop_error : BOOL;

	DesludgePump_P201B_1_overload_Filter : ErrorFilter;
	DesludgePump_P201B_1_incomplete_Filter : ErrorFilter;
	DesludgePump_P201B_1_status_Filter : ErrorFilter;
	DesludgePump_P201B_1_stop_Filter : ErrorFilter;



	DesludgePump_P201B_2_remote_mode AT%I* : BOOL;
	DesludgePump_P201B_2_overload AT%I* : BOOL;
	DesludgePump_P201B_2_incomplete AT%I* : BOOL;
	DesludgePump_P201B_2_status AT%I* : BOOL;

	DesludgePump_P201B_2_command AT%Q* : BOOL;

	DesludgePump_P201B_2_in : BOOL;
	DesludgePump_P201B_2_overload_error : BOOL;
	DesludgePump_P201B_2_incomplete_error : BOOL;
	DesludgePump_P201B_2_status_error : BOOL;
	DesludgePump_P201B_2_common_error : BOOL;
	DesludgePump_P201B_2_stop_error : BOOL;

	DesludgePump_P201B_2_overload_Filter : ErrorFilter;
	DesludgePump_P201B_2_incomplete_Filter : ErrorFilter;
	DesludgePump_P201B_2_status_Filter : ErrorFilter;
	DesludgePump_P201B_2_stop_Filter : ErrorFilter;

	DesludgePump_P201B :Equipment_Dual;


	Blower_B201B_1_remote_mode AT%I* : BOOL;
	Blower_B201B_1_overload AT%I* : BOOL;
	Blower_B201B_1_incomplete AT%I* : BOOL;
	Blower_B201B_1_status AT%I* : BOOL;

	Blower_B201B_1_command AT%Q* : BOOL;

	Blower_B201B_1_in : BOOL;
	Blower_B201B_1_overload_error : BOOL;
	Blower_B201B_1_incomplete_error : BOOL;
	Blower_B201B_1_status_error : BOOL;
	Blower_B201B_1_common_error : BOOL;
	Blower_B201B_1_stop_error : BOOL;

	Blower_B201B_1_overload_Filter : ErrorFilter;
	Blower_B201B_1_incomplete_Filter : ErrorFilter;
	Blower_B201B_1_status_Filter : ErrorFilter;
	Blower_B201B_1_stop_Filter : ErrorFilter;



	Blower_B201B_2_remote_mode AT%I* : BOOL;
	Blower_B201B_2_overload AT%I* : BOOL;
	Blower_B201B_2_incomplete AT%I* : BOOL;
	Blower_B201B_2_status AT%I* : BOOL;

	Blower_B201B_2_command AT%Q* : BOOL;

	Blower_B201B_2_in : BOOL;
	Blower_B201B_2_overload_error : BOOL;
	Blower_B201B_2_incomplete_error : BOOL;
	Blower_B201B_2_status_error : BOOL;
	Blower_B201B_2_common_error : BOOL;
	Blower_B201B_2_stop_error : BOOL;

	Blower_B201B_2_overload_Filter : ErrorFilter;
	Blower_B201B_2_incomplete_Filter : ErrorFilter;
	Blower_B201B_2_status_Filter : ErrorFilter;
	Blower_B201B_2_stop_Filter : ErrorFilter;



	Blower_B201B_3_remote_mode AT%I* : BOOL;
	Blower_B201B_3_overload AT%I* : BOOL;
	Blower_B201B_3_incomplete AT%I* : BOOL;
	Blower_B201B_3_status AT%I* : BOOL;

	Blower_B201B_3_command AT%Q* : BOOL;

	Blower_B201B_3_in : BOOL;
	Blower_B201B_3_overload_error : BOOL;
	Blower_B201B_3_incomplete_error : BOOL;
	Blower_B201B_3_status_error : BOOL;
	Blower_B201B_3_common_error : BOOL;
	Blower_B201B_3_stop_error : BOOL;

	Blower_B201B_3_overload_Filter : ErrorFilter;
	Blower_B201B_3_incomplete_Filter : ErrorFilter;
	Blower_B201B_3_status_Filter : ErrorFilter;
	Blower_B201B_3_stop_Filter : ErrorFilter;


END_VAR

VAR PERSISTENT
	FILLING_TOKEN : INT;
	AERATION_TOKEN: INT;
	DECANTING_TOKEN: INT;
END_VAR
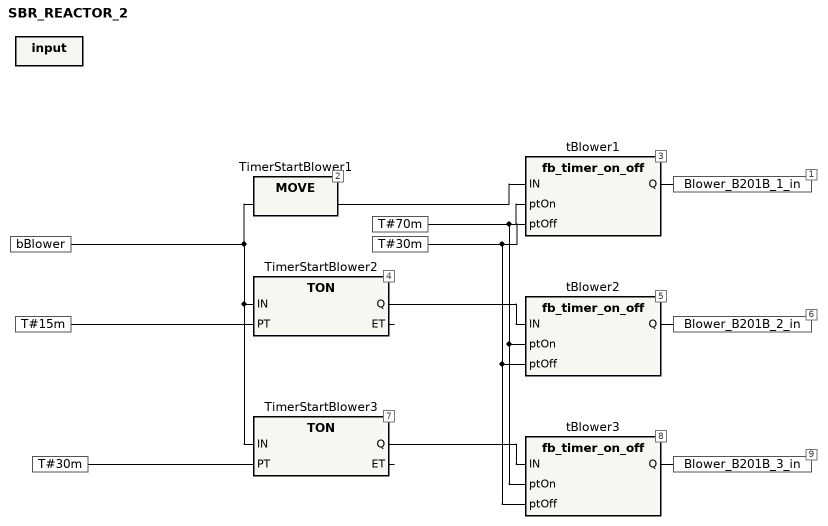
_CFC_ (* Continuous Function Chart, elements in execution order *)
#0 input()
#1 Blower_B201B_1_in <= #3.Q
#2 TimerStartBlower1:MOVE(bBlower)
#3 tBlower1:fb_timer_on_off(IN: #2, ptOn: T#70m, ptOff: T#30m)
#4 TimerStartBlower2:TON(IN: bBlower, PT: T#15m)
#5 tBlower2:fb_timer_on_off(IN: #4.Q, ptOn: T#70m, ptOff: T#30m)
#6 Blower_B201B_2_in <= #5.Q
#7 TimerStartBlower3:TON(IN: bBlower, PT: T#30m)
#8 tBlower3:fb_timer_on_off(IN: #7.Q, ptOn: T#70m, ptOff: T#30m)
#9 Blower_B201B_3_in <= #8.Q
_END_CFC_
END_PROGRAM
ACTION input:
SludeTankSensorLevelHi_LSL510B();

SBRReactor_1(
	bEnable:=SBR_B_1_bEnable_SW ,
	SludgeTankLevelHi:= SludeTankSensorLevelHi_LSL510B.Q,
	SBRLevelSensor_LSH200:= SBR_B_1_SBRLevelSensor_LSH200,
	rDO201:= SBR_B_1_DOSensor_DO201,
	DecanterLevelSensorHi:=SBR_B_1_DecanterLevelSensorHi_Rx ,
	DecanterLevelSensorLow:=SBR_B_1_DecanterLevelSensorLow_Rx ,
	FILLING_TOKEN:=FILLING_TOKEN ,
	AERATION_TOKEN:= AERATION_TOKEN,
	DECANTING_TOKEN:= DECANTING_TOKEN,
	bBlowerOn=>SBR_B_1_Blower_B201 ,
	bDeSludgePump=>SBR_B_1_DesludgePump_P201 ,
	bFilling=>SBR_B_1_filling ,
	bAeration=>SBR_B_1_aeration ,
	bSettling=>SBR_B_1_settling ,
	bDecanting=>SBR_B_1_decanting ,
	bDesluging=>SBR_B_1_desludging ,
	bWarning_DoNotInRange=>SBR_B_1_warning_DONotInRange ,
	bForwardDecant=>SBR_B_1_FowardDecant_XV26 ,
	bReverseDecant=>SBR_B_1_ReverseDecant_XV26 ,
	bBlowerValve_XV201=>SBR_B_1_BlowerValve_XV201 ,
	bDeslugValve_XV241=> SBR_B_1_DeSludgeValve_XV241,
	bSBRValve_XV205=>SBR_B_1_SBRValve_XV205 ,
	bSBRMixer=>SBR_B_1_SBRMixer_XV205 );


SBRReactor_2(
	bEnable:=SBR_B_2_bEnable_SW ,
	SludgeTankLevelHi:= SludeTankSensorLevelHi_LSL510B.Q,
	SBRLevelSensor_LSH200:= SBR_B_2_SBRLevelSensor_LSH200,
	rDO201:= SBR_B_2_DOSensor_DO201,
	DecanterLevelSensorHi:=SBR_B_2_DecanterLevelSensorHi_Rx ,
	DecanterLevelSensorLow:=SBR_B_2_DecanterLevelSensorLow_Rx ,
	FILLING_TOKEN:=FILLING_TOKEN ,
	AERATION_TOKEN:= AERATION_TOKEN,
	DECANTING_TOKEN:= DECANTING_TOKEN,
	bBlowerOn=>SBR_B_2_Blower_B201 ,
	bDeSludgePump=>SBR_B_2_DesludgePump_P201 ,
	bFilling=>SBR_B_2_filling ,
	bAeration=>SBR_B_2_aeration ,
	bSettling=>SBR_B_2_settling ,
	bDecanting=>SBR_B_2_decanting ,
	bDesluging=>SBR_B_2_desludging ,
	bWarning_DoNotInRange=>SBR_B_2_warning_DONotInRange ,
	bForwardDecant=>SBR_B_2_FowardDecant_XV26 ,
	bReverseDecant=>SBR_B_2_ReverseDecant_XV26 ,
	bBlowerValve_XV201=>SBR_B_2_BlowerValve_XV201 ,
	bDeslugValve_XV241=> SBR_B_2_DeSludgeValve_XV241,
	bSBRValve_XV205=>SBR_B_2_SBRValve_XV205 ,
	bSBRMixer=>SBR_B_2_SBRMixer_XV205 );


SBRReactor_3(
	bEnable:=SBR_B_3_bEnable_SW ,
	SludgeTankLevelHi:= SludeTankSensorLevelHi_LSL510B.Q,
	SBRLevelSensor_LSH200:= SBR_B_3_SBRLevelSensor_LSH200,
	rDO201:= SBR_B_3_DOSensor_DO201,
	DecanterLevelSensorHi:=SBR_B_3_DecanterLevelSensorHi_Rx ,
	DecanterLevelSensorLow:=SBR_B_3_DecanterLevelSensorLow_Rx ,
	FILLING_TOKEN:=FILLING_TOKEN ,
	AERATION_TOKEN:= AERATION_TOKEN,
	DECANTING_TOKEN:= DECANTING_TOKEN,
	bBlowerOn=>SBR_B_3_Blower_B201 ,
	bDeSludgePump=>SBR_B_3_DesludgePump_P201 ,
	bFilling=>SBR_B_3_filling ,
	bAeration=>SBR_B_3_aeration ,
	bSettling=>SBR_B_3_settling ,
	bDecanting=>SBR_B_3_decanting ,
	bDesluging=>SBR_B_3_desludging ,
	bWarning_DoNotInRange=>SBR_B_3_warning_DONotInRange ,
	bForwardDecant=>SBR_B_3_FowardDecant_XV26 ,
	bReverseDecant=>SBR_B_3_ReverseDecant_XV26 ,
	bBlowerValve_XV201=>SBR_B_3_BlowerValve_XV201 ,
	bDeslugValve_XV241=> SBR_B_3_DeSludgeValve_XV241,
	bSBRValve_XV205=>SBR_B_3_SBRValve_XV205 ,
	bSBRMixer=>SBR_B_3_SBRMixer_XV205 );


SBRReactor_4(
	bEnable:=SBR_B_4_bEnable_SW ,
	SludgeTankLevelHi:= SludeTankSensorLevelHi_LSL510B.Q,
	SBRLevelSensor_LSH200:= SBR_B_4_SBRLevelSensor_LSH200,
	rDO201:= SBR_B_4_DOSensor_DO201,
	DecanterLevelSensorHi:=SBR_B_4_DecanterLevelSensorHi_Rx ,
	DecanterLevelSensorLow:=SBR_B_4_DecanterLevelSensorLow_Rx ,
	FILLING_TOKEN:=FILLING_TOKEN ,
	AERATION_TOKEN:= AERATION_TOKEN,
	DECANTING_TOKEN:= DECANTING_TOKEN,
	bBlowerOn=>SBR_B_4_Blower_B201 ,
	bDeSludgePump=>SBR_B_4_DesludgePump_P201 ,
	bFilling=>SBR_B_4_filling ,
	bAeration=>SBR_B_4_aeration ,
	bSettling=>SBR_B_4_settling ,
	bDecanting=>SBR_B_4_decanting ,
	bDesluging=>SBR_B_4_desludging ,
	bWarning_DoNotInRange=>SBR_B_4_warning_DONotInRange ,
	bForwardDecant=>SBR_B_4_FowardDecant_XV26 ,
	bReverseDecant=>SBR_B_4_ReverseDecant_XV26 ,
	bBlowerValve_XV201=>SBR_B_4_BlowerValve_XV201 ,
	bDeslugValve_XV241=> SBR_B_4_DeSludgeValve_XV241,
	bSBRValve_XV205=>SBR_B_4_SBRValve_XV205 ,
	bSBRMixer=>SBR_B_4_SBRMixer_XV205 );


bDeSludge:=SBR_B_1_DeSludgeValve_XV241 OR SBR_B_2_DeSludgeValve_XV241 OR SBR_B_3_DeSludgeValve_XV241 OR SBR_B_4_DeSludgeValve_XV241;
bBlower:= SBR_B_1_Blower_B201 OR SBR_B_2_Blower_B201 OR SBR_B_3_Blower_B201 OR SBR_B_4_Blower_B201;



SBRMixer_M200B1_A_in := SBR_B_1_SBRMixer_XV205;
SBRMixer_M200B1_A_command := SBRMixer_M200B1_A_in AND SBRMixer_M200B1_A_remote_mode;
SBRMixer_M200B1_A_overload_Filter(IN:=(SBRMixer_M200B1_A_overload AND SBRMixer_M200B1_A_in),PT:=T#2s,Q=>SBRMixer_M200B1_A_overload_error);
SBRMixer_M200B1_A_incomplete_Filter(IN:=(SBRMixer_M200B1_A_incomplete AND SBRMixer_M200B1_A_in),PT:=T#2s,Q=>SBRMixer_M200B1_A_incomplete_error);
SBRMixer_M200B1_A_status_Filter(IN:=(NOT SBRMixer_M200B1_A_status AND SBRMixer_M200B1_A_in),PT:=T#10s, Q=>SBRMixer_M200B1_A_status_error);
SBRMixer_M200B1_A_stop_Filter(IN:=( SBRMixer_M200B1_A_status AND NOT SBRMixer_M200B1_A_in),PT:=T#10s, Q=>SBRMixer_M200B1_A_stop_error);

SBRMixer_M200B1_A_common_error := SBRMixer_M200B1_A_overload_error OR SBRMixer_M200B1_A_incomplete_error OR SBRMixer_M200B1_A_status_error OR SBRMixer_M200B1_A_stop_error;


SBRMixer_M200B1_B_in := SBR_B_1_SBRMixer_XV205;
SBRMixer_M200B1_B_command := SBRMixer_M200B1_B_in AND SBRMixer_M200B1_B_remote_mode;
SBRMixer_M200B1_B_overload_Filter(IN:=(SBRMixer_M200B1_B_overload AND SBRMixer_M200B1_B_in),PT:=T#2s,Q=>SBRMixer_M200B1_B_overload_error);
SBRMixer_M200B1_B_incomplete_Filter(IN:=(SBRMixer_M200B1_B_incomplete AND SBRMixer_M200B1_B_in),PT:=T#2s,Q=>SBRMixer_M200B1_B_incomplete_error);
SBRMixer_M200B1_B_status_Filter(IN:=(NOT SBRMixer_M200B1_B_status AND SBRMixer_M200B1_B_in),PT:=T#10s, Q=>SBRMixer_M200B1_B_status_error);
SBRMixer_M200B1_B_stop_Filter(IN:=( SBRMixer_M200B1_B_status AND NOT SBRMixer_M200B1_B_in),PT:=T#10s, Q=>SBRMixer_M200B1_B_stop_error);

SBRMixer_M200B1_B_common_error := SBRMixer_M200B1_B_overload_error OR SBRMixer_M200B1_B_incomplete_error OR SBRMixer_M200B1_B_status_error OR SBRMixer_M200B1_B_stop_error;


SBRMixer_M200B1_C_in := SBR_B_1_SBRMixer_XV205;
SBRMixer_M200B1_C_command := SBRMixer_M200B1_C_in AND SBRMixer_M200B1_C_remote_mode;
SBRMixer_M200B1_C_overload_Filter(IN:=(SBRMixer_M200B1_C_overload AND SBRMixer_M200B1_C_in),PT:=T#2s,Q=>SBRMixer_M200B1_C_overload_error);
SBRMixer_M200B1_C_incomplete_Filter(IN:=(SBRMixer_M200B1_C_incomplete AND SBRMixer_M200B1_C_in),PT:=T#2s,Q=>SBRMixer_M200B1_C_incomplete_error);
SBRMixer_M200B1_C_status_Filter(IN:=(NOT SBRMixer_M200B1_C_status AND SBRMixer_M200B1_C_in),PT:=T#10s, Q=>SBRMixer_M200B1_C_status_error);
SBRMixer_M200B1_C_stop_Filter(IN:=( SBRMixer_M200B1_C_status AND NOT SBRMixer_M200B1_C_in),PT:=T#10s, Q=>SBRMixer_M200B1_C_stop_error);

SBRMixer_M200B1_C_common_error := SBRMixer_M200B1_C_overload_error OR SBRMixer_M200B1_C_incomplete_error OR SBRMixer_M200B1_C_status_error OR SBRMixer_M200B1_C_stop_error;



SBRMixer_M200B2_A_in := SBR_B_2_SBRMixer_XV205;
SBRMixer_M200B2_A_command := SBRMixer_M200B2_A_in AND SBRMixer_M200B2_A_remote_mode;
SBRMixer_M200B2_A_overload_Filter(IN:=(SBRMixer_M200B2_A_overload AND SBRMixer_M200B2_A_in),PT:=T#2s,Q=>SBRMixer_M200B2_A_overload_error);
SBRMixer_M200B2_A_incomplete_Filter(IN:=(SBRMixer_M200B2_A_incomplete AND SBRMixer_M200B2_A_in),PT:=T#2s,Q=>SBRMixer_M200B2_A_incomplete_error);
SBRMixer_M200B2_A_status_Filter(IN:=(NOT SBRMixer_M200B2_A_status AND SBRMixer_M200B2_A_in),PT:=T#10s, Q=>SBRMixer_M200B2_A_status_error);
SBRMixer_M200B2_A_stop_Filter(IN:=( SBRMixer_M200B2_A_status AND NOT SBRMixer_M200B2_A_in),PT:=T#10s, Q=>SBRMixer_M200B2_A_stop_error);

SBRMixer_M200B2_A_common_error := SBRMixer_M200B2_A_overload_error OR SBRMixer_M200B2_A_incomplete_error OR SBRMixer_M200B2_A_status_error OR SBRMixer_M200B2_A_stop_error;


SBRMixer_M200B2_B_in := SBR_B_2_SBRMixer_XV205;
SBRMixer_M200B2_B_command := SBRMixer_M200B2_B_in AND SBRMixer_M200B2_B_remote_mode;
SBRMixer_M200B2_B_overload_Filter(IN:=(SBRMixer_M200B2_B_overload AND SBRMixer_M200B2_B_in),PT:=T#2s,Q=>SBRMixer_M200B2_B_overload_error);
SBRMixer_M200B2_B_incomplete_Filter(IN:=(SBRMixer_M200B2_B_incomplete AND SBRMixer_M200B2_B_in),PT:=T#2s,Q=>SBRMixer_M200B2_B_incomplete_error);
SBRMixer_M200B2_B_status_Filter(IN:=(NOT SBRMixer_M200B2_B_status AND SBRMixer_M200B2_B_in),PT:=T#10s, Q=>SBRMixer_M200B2_B_status_error);
SBRMixer_M200B1_B_stop_Filter(IN:=( SBRMixer_M200B1_B_status AND NOT SBRMixer_M200B1_B_in),PT:=T#10s, Q=>SBRMixer_M200B1_B_stop_error);

SBRMixer_M200B1_B_common_error := SBRMixer_M200B1_B_overload_error OR SBRMixer_M200B1_B_incomplete_error OR SBRMixer_M200B1_B_status_error OR SBRMixer_M200B1_B_stop_error;


SBRMixer_M200B2_C_in := SBR_B_2_SBRMixer_XV205;
SBRMixer_M200B2_C_command := SBRMixer_M200B2_C_in AND SBRMixer_M200B2_C_remote_mode;
SBRMixer_M200B2_C_overload_Filter(IN:=(SBRMixer_M200B2_C_overload AND SBRMixer_M200B2_C_in),PT:=T#2s,Q=>SBRMixer_M200B2_C_overload_error);
SBRMixer_M200B2_C_incomplete_Filter(IN:=(SBRMixer_M200B2_C_incomplete AND SBRMixer_M200B2_C_in),PT:=T#2s,Q=>SBRMixer_M200B2_C_incomplete_error);
SBRMixer_M200B2_C_status_Filter(IN:=(NOT SBRMixer_M200B2_C_status AND SBRMixer_M200B2_C_in),PT:=T#10s, Q=>SBRMixer_M200B2_C_status_error);
SBRMixer_M200B2_C_stop_Filter(IN:=( SBRMixer_M200B2_C_status AND NOT SBRMixer_M200B2_C_in),PT:=T#10s, Q=>SBRMixer_M200B2_C_stop_error);

SBRMixer_M200B2_C_common_error := SBRMixer_M200B2_C_overload_error OR SBRMixer_M200B2_C_incomplete_error OR SBRMixer_M200B2_C_status_error OR SBRMixer_M200B2_C_stop_error;



SBRMixer_M200B3_A_in := SBR_B_3_SBRMixer_XV205;
SBRMixer_M200B3_A_command := SBRMixer_M200B3_A_in AND SBRMixer_M200B3_A_remote_mode;
SBRMixer_M200B3_A_overload_Filter(IN:=(SBRMixer_M200B3_A_overload AND SBRMixer_M200B3_A_in),PT:=T#2s,Q=>SBRMixer_M200B3_A_overload_error);
SBRMixer_M200B3_A_incomplete_Filter(IN:=(SBRMixer_M200B3_A_incomplete AND SBRMixer_M200B3_A_in),PT:=T#2s,Q=>SBRMixer_M200B3_A_incomplete_error);
SBRMixer_M200B3_A_status_Filter(IN:=(NOT SBRMixer_M200B3_A_status AND SBRMixer_M200B3_A_in),PT:=T#10s, Q=>SBRMixer_M200B3_A_status_error);
SBRMixer_M200B3_A_stop_Filter(IN:=( SBRMixer_M200B3_A_status AND NOT SBRMixer_M200B3_A_in),PT:=T#10s, Q=>SBRMixer_M200B3_A_stop_error);

SBRMixer_M200B3_A_common_error := SBRMixer_M200B3_A_overload_error OR SBRMixer_M200B3_A_incomplete_error OR SBRMixer_M200B3_A_status_error OR SBRMixer_M200B3_A_stop_error;


SBRMixer_M200B3_B_in := SBR_B_3_SBRMixer_XV205;
SBRMixer_M200B3_B_command := SBRMixer_M200B3_B_in AND SBRMixer_M200B3_B_remote_mode;
SBRMixer_M200B3_B_overload_Filter(IN:=(SBRMixer_M200B3_B_overload AND SBRMixer_M200B3_B_in),PT:=T#2s,Q=>SBRMixer_M200B3_B_overload_error);
SBRMixer_M200B3_B_incomplete_Filter(IN:=(SBRMixer_M200B3_B_incomplete AND SBRMixer_M200B3_B_in),PT:=T#2s,Q=>SBRMixer_M200B3_B_incomplete_error);
SBRMixer_M200B3_B_status_Filter(IN:=(NOT SBRMixer_M200B3_B_status AND SBRMixer_M200B3_B_in),PT:=T#10s, Q=>SBRMixer_M200B3_B_status_error);
SBRMixer_M200B1_B_stop_Filter(IN:=( SBRMixer_M200B1_B_status AND NOT SBRMixer_M200B1_B_in),PT:=T#10s, Q=>SBRMixer_M200B1_B_stop_error);

SBRMixer_M200B1_B_common_error := SBRMixer_M200B1_B_overload_error OR SBRMixer_M200B1_B_incomplete_error OR SBRMixer_M200B1_B_status_error OR SBRMixer_M200B1_B_stop_error;


SBRMixer_M200B3_C_in := SBR_B_3_SBRMixer_XV205;
SBRMixer_M200B3_C_command := SBRMixer_M200B3_C_in AND SBRMixer_M200B3_C_remote_mode;
SBRMixer_M200B3_C_overload_Filter(IN:=(SBRMixer_M200B3_C_overload AND SBRMixer_M200B3_C_in),PT:=T#2s,Q=>SBRMixer_M200B3_C_overload_error);
SBRMixer_M200B3_C_incomplete_Filter(IN:=(SBRMixer_M200B3_C_incomplete AND SBRMixer_M200B3_C_in),PT:=T#2s,Q=>SBRMixer_M200B3_C_incomplete_error);
SBRMixer_M200B3_C_status_Filter(IN:=(NOT SBRMixer_M200B3_C_status AND SBRMixer_M200B3_C_in),PT:=T#10s, Q=>SBRMixer_M200B3_C_status_error);
SBRMixer_M200B3_C_stop_Filter(IN:=( SBRMixer_M200B3_C_status AND NOT SBRMixer_M200B3_C_in),PT:=T#10s, Q=>SBRMixer_M200B3_C_stop_error);

SBRMixer_M200B3_C_common_error := SBRMixer_M200B3_C_overload_error OR SBRMixer_M200B3_C_incomplete_error OR SBRMixer_M200B3_C_status_error OR SBRMixer_M200B3_C_stop_error;



DesludgePump_P201B_1_overload_Filter(IN:=(DesludgePump_P201B_1_overload AND DesludgePump_P201B_1_in),PT:=T#2s,Q=>DesludgePump_P201B_1_overload_error);
DesludgePump_P201B_1_incomplete_Filter(IN:=(DesludgePump_P201B_1_incomplete AND DesludgePump_P201B_1_in),PT:=T#2s,Q=>DesludgePump_P201B_1_incomplete_error);
DesludgePump_P201B_1_status_Filter(IN:=(NOT DesludgePump_P201B_1_status AND DesludgePump_P201B_1_in),PT:=T#10s, Q=>DesludgePump_P201B_1_status_error);
DesludgePump_P201B_1_stop_Filter(IN:=( DesludgePump_P201B_1_status AND NOT DesludgePump_P201B_1_in),PT:=T#10s, Q=>DesludgePump_P201B_1_stop_error);

DesludgePump_P201B_1_common_error := DesludgePump_P201B_1_overload_error OR DesludgePump_P201B_1_incomplete_error OR DesludgePump_P201B_1_status_error OR DesludgePump_P201B_1_stop_error;


DesludgePump_P201B_2_overload_Filter(IN:=(DesludgePump_P201B_2_overload AND DesludgePump_P201B_2_in),PT:=T#2s,Q=>DesludgePump_P201B_2_overload_error);
DesludgePump_P201B_2_incomplete_Filter(IN:=(DesludgePump_P201B_2_incomplete AND DesludgePump_P201B_2_in),PT:=T#2s,Q=>DesludgePump_P201B_2_incomplete_error);
DesludgePump_P201B_2_status_Filter(IN:=(NOT DesludgePump_P201B_2_status AND DesludgePump_P201B_2_in),PT:=T#10s, Q=>DesludgePump_P201B_2_status_error);
DesludgePump_P201B_2_stop_Filter(IN:=( DesludgePump_P201B_2_status AND NOT DesludgePump_P201B_2_in),PT:=T#10s, Q=>DesludgePump_P201B_2_stop_error);

DesludgePump_P201B_2_common_error := DesludgePump_P201B_2_overload_error OR DesludgePump_P201B_2_incomplete_error OR DesludgePump_P201B_2_status_error OR DesludgePump_P201B_2_stop_error;

DesludgePump_P201B_1_in := bDeSludge;
DesludgePump_P201B(
	ERROR1:=DesludgePump_P201B_1_common_error ,
	ERROR2:=DesludgePump_P201B_2_common_error ,
	remote1:=DesludgePump_P201B_1_remote_mode ,
	remote2:=DesludgePump_P201B_2_remote_mode ,
	IN1:=DesludgePump_P201B_1_in ,
	IN2:=DesludgePump_P201B_2_in ,
	Command1=>DesludgePump_P201B_1_command,
	Command2=>DesludgePump_P201B_2_command );


Blower_B201B_1_command := Blower_B201B_1_in AND Blower_B201B_1_remote_mode;
Blower_B201B_1_overload_Filter(IN:=(Blower_B201B_1_overload AND Blower_B201B_1_in),PT:=T#2s,Q=>Blower_B201B_1_overload_error);
Blower_B201B_1_incomplete_Filter(IN:=(Blower_B201B_1_incomplete AND Blower_B201B_1_in),PT:=T#2s,Q=>Blower_B201B_1_incomplete_error);
Blower_B201B_1_status_Filter(IN:=(NOT Blower_B201B_1_status AND Blower_B201B_1_in),PT:=T#10s, Q=>Blower_B201B_1_status_error);
Blower_B201B_1_stop_Filter(IN:=( Blower_B201B_1_status AND NOT Blower_B201B_1_in),PT:=T#10s, Q=>Blower_B201B_1_stop_error);

Blower_B201B_1_common_error := Blower_B201B_1_overload_error OR Blower_B201B_1_incomplete_error OR Blower_B201B_1_status_error OR Blower_B201B_1_stop_error;


Blower_B201B_2_command := Blower_B201B_2_in AND Blower_B201B_2_remote_mode;
Blower_B201B_2_overload_Filter(IN:=(Blower_B201B_2_overload AND Blower_B201B_2_in),PT:=T#2s,Q=>Blower_B201B_2_overload_error);
Blower_B201B_2_incomplete_Filter(IN:=(Blower_B201B_2_incomplete AND Blower_B201B_2_in),PT:=T#2s,Q=>Blower_B201B_2_incomplete_error);
Blower_B201B_2_status_Filter(IN:=(NOT Blower_B201B_2_status AND Blower_B201B_2_in),PT:=T#10s, Q=>Blower_B201B_2_status_error);
Blower_B201B_2_stop_Filter(IN:=( Blower_B201B_2_status AND NOT Blower_B201B_2_in),PT:=T#10s, Q=>Blower_B201B_2_stop_error);

Blower_B201B_2_common_error := Blower_B201B_2_overload_error OR Blower_B201B_2_incomplete_error OR Blower_B201B_2_status_error OR Blower_B201B_2_stop_error;


Blower_B201B_3_command := Blower_B201B_3_in AND Blower_B201B_3_remote_mode;
Blower_B201B_3_overload_Filter(IN:=(Blower_B201B_3_overload AND Blower_B201B_3_in),PT:=T#2s,Q=>Blower_B201B_3_overload_error);
Blower_B201B_3_incomplete_Filter(IN:=(Blower_B201B_3_incomplete AND Blower_B201B_3_in),PT:=T#2s,Q=>Blower_B201B_3_incomplete_error);
Blower_B201B_3_status_Filter(IN:=(NOT Blower_B201B_3_status AND Blower_B201B_3_in),PT:=T#10s, Q=>Blower_B201B_3_status_error);
Blower_B201B_3_stop_Filter(IN:=( Blower_B201B_3_status AND NOT Blower_B201B_3_in),PT:=T#10s, Q=>Blower_B201B_3_stop_error);

Blower_B201B_3_common_error := Blower_B201B_3_overload_error OR Blower_B201B_3_incomplete_error OR Blower_B201B_3_status_error OR Blower_B201B_3_stop_error;
END_ACTION

(* POU module/fb_timer_on_off, CFC *)
FUNCTION_BLOCK fb_timer_on_off
VAR_INPUT
	IN: BOOL;
	ptOn: TIME;
	ptOff: TIME;
END_VAR
VAR_OUTPUT
	Q: BOOL;
END_VAR
VAR
	ON: TON;
	OFF: TON;
END_VAR
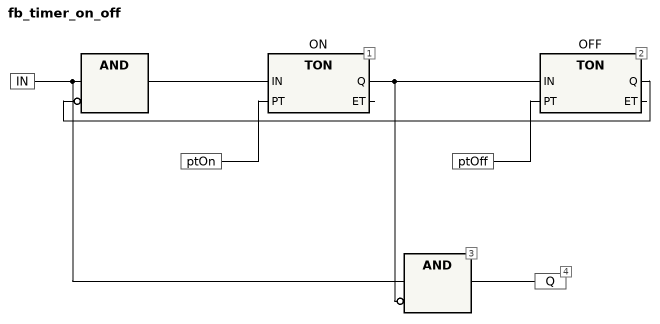
_CFC_ (* Continuous Function Chart, elements in execution order *)
#0 AND(IN, NOT #2.Q)
#1 ON:TON(IN: #0, PT: ptOn)
#2 OFF:TON(IN: #1.Q, PT: ptOff)
#3 AND(IN, NOT #1.Q)
#4 Q <= #3
_END_CFC_
(* the same logic as Structured Text *)
ON(IN := IN AND NOT OFF.Q, PT := ptOn);
OFF(IN := ON.Q, PT := ptOff);
Q := IN AND NOT ON.Q;
END_FUNCTION_BLOCK

(* POU module/SBRReactor, ST *)
FUNCTION_BLOCK SBRReactor
VAR_INPUT
	bEnable : BOOL;
	SludgeTankLevelHi: BOOL;
	SBRLevelSensor_LSH200: BOOL;
	rDO201: INT;
	DecanterLevelSensorHi : BOOL;
	DecanterLevelSensorLow : BOOL;

END_VAR
VAR_OUTPUT

	bBlowerOn: BOOL;
	bDeSludgePump: BOOL;


	bFilling: BOOL;
	bAeration: BOOL;
	bSettling: BOOL;
	bDecanting: BOOL;
	bDesluging: BOOL;



	bForwardDecant : BOOL;
	bReverseDecant: BOOL;
	bBlowerValve_XV201 : BOOL;
	bDeslugValve_XV241: BOOL;
	bSBRValve_XV205 : BOOL;

	bSBRMixer: BOOL;

	bWarning_DoNotInRange: BOOL;
END_VAR
VAR PERSISTENT
	step: INT;
END_VAR
VAR
	bFillingDone: BOOL;
	bAerationDone: BOOL;
	bSettingDone: BOOL;
	bDecantingDone: BOOL;


	decant: INT;
	MixerOff: TON;
	timerBlower: TON;
	DOtimer: TON;
	TimerSettling: TON;
	timerDecant: TON;
	DecantTimeLapse: TON;
END_VAR

VAR_IN_OUT
	FILLING_TOKEN : INT;
	AERATION_TOKEN: INT;
	DECANTING_TOKEN: INT;
END_VAR
VAR (* helpers for the ST form of the networks *)
	_en12 : BOOL;
	_t12 : BOOL;
END_VAR
bFilling:= FALSE;
bAeration:= FALSE;
bSettling:= FALSE;
bDecanting:= FALSE;

IF NOT bEnable THEN
	step := 0;
END_IF

CASE step OF
0:
	(*Idle*)
	step := 10;
10:

	IF FILLING_TOKEN > 0 THEN
		FILLING_TOKEN :=0;
		step := 15;
	END_IF
15:
	bFilling :=TRUE;
	IF bFillingDone THEN
		step := 20;
		FILLING_TOKEN := 1;
	END_IF
20:

	IF AERATION_TOKEN > 0 THEN
		step := 25;
		AERATION_TOKEN := 0;
	END_IF
25:
	IF bAerationDone THEN
		step:= 30;
		AERATION_TOKEN := 1;
	END_IF
30:
	bSettling := TRUE;
	IF bSettingDone THEN
		step := 40;
	END_IF
40:
	IF DECANTING_TOKEN > 0 THEN
		DECANTING_TOKEN := 0;
		step := 45;
	END_IF
45:
		bDecanting := TRUE;
		IF bDecantingDone THEN
			step := 0;
			DECANTING_TOKEN := 1;
		END_IF
END_CASE



filling;
Aeration;
Settle;
Decanting;
END_FUNCTION_BLOCK
ACTION Aeration:
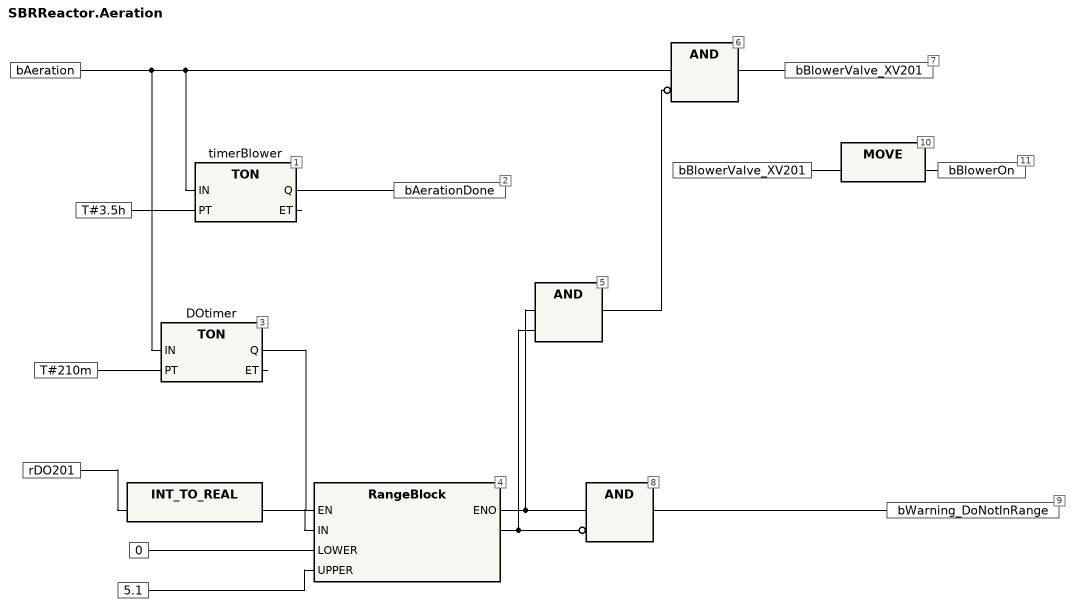
_CFC_ (* Continuous Function Chart, elements in execution order *)
#0 INT_TO_REAL(rDO201)
#1 timerBlower:TON(IN: bAeration, PT: T#3.5h)
#2 bAerationDone <= #1.Q
#3 DOtimer:TON(IN: bAeration, PT: T#210m)
#4 RangeBlock(EN: #3.Q, IN: #0, LOWER: 0, UPPER: 5.1)
#5 AND(#4.ENO, #4)
#6 AND(bAeration, NOT #5)
#7 bBlowerValve_XV201 <= #6
#8 AND(#4.ENO, NOT #4)
#9 bWarning_DoNotInRange <= #8
#10 MOVE(bBlowerValve_XV201)
#11 bBlowerOn <= #10
_END_CFC_
(* the same logic as Structured Text *)
timerBlower(IN := bAeration, PT := T#3.5h);
bAerationDone := timerBlower.Q;
DOtimer(IN := bAeration, PT := T#210m);
_en12 := DOtimer.Q;
IF _en12 THEN _t12 := RangeBlock(IN := INT_TO_REAL(rDO201), LOWER := 0, UPPER := 5.1); END_IF;
bBlowerValve_XV201 := bAeration AND NOT (_en12 AND _t12);
bWarning_DoNotInRange := _en12 AND NOT _t12;
bBlowerOn := bBlowerValve_XV201;
END_ACTION
ACTION Decanting:
IF NOT bDecanting THEN
decant := 0;
END_IF

bDecantingDone := (decant >= 60);


CASE decant OF
0:
	decant := 10;
10:

	IF DecanterLevelSensorHi THEN
		(*start Reverse Sequence*)
		bForwardDecant :=FALSE;
		decant := 20;
	ELSE
		bForwardDecant :=TRUE;
	END_IF


20:
	bReverseDecant := TRUE;
	timerDecant(IN:= TRUE, PT:= T#2s);
		IF timerDecant.Q THEN
			timerDecant(IN:= FALSE);
			bReverseDecant := FALSE;
			decant := 30;
		END_IF
30:
	timerDecant(IN:= TRUE, PT:= T#10s);
		IF timerDecant.Q THEN
			timerDecant(IN:= FALSE);
			IF DecanterLevelSensorLow THEN
				decant := 40;
			ELSE
				decant := 20;
			END_IF
		END_IF
40:
	timerDecant(IN:=TRUE,PT:=T#300s);
	IF timerDecant.Q THEN
		timerDecant(IN:=FALSE);
		decant := 50;
	END_IF
50:

	IF DecanterLevelSensorHi THEN
		(*start Reverse Sequence*)
		bForwardDecant :=FALSE;
		decant := 60;
	ELSE
		bForwardDecant :=TRUE;
	END_IF
60:
;
END_CASE

DecantTimeLapse(IN:=bDecanting, PT:= T#4000s);
bDesluging := (DecantTimeLapse.ET <= T#15m) OR (DecantTimeLapse.ET >= T#15m);

bDeslugValve_XV241 := bDesluging AND NOT SludgeTankLevelHi;
bDeSludgePump := bDeslugValve_XV241;
END_ACTION
ACTION filling:
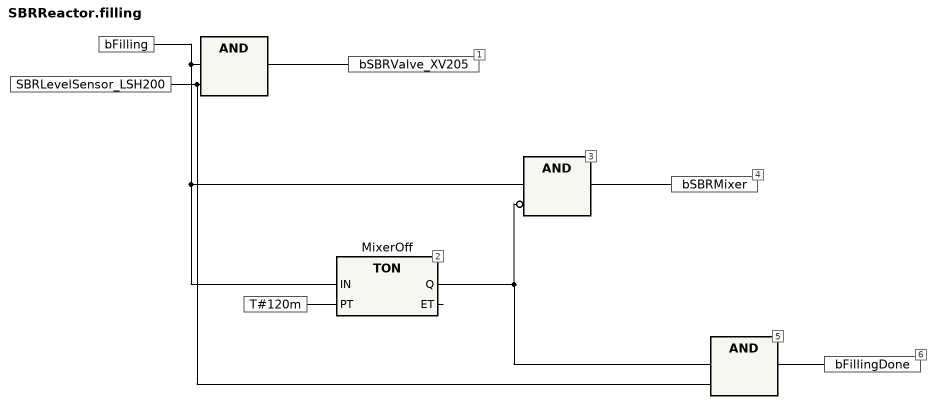
_CFC_ (* Continuous Function Chart, elements in execution order *)
#0 AND(bFilling, SBRLevelSensor_LSH200)
#1 bSBRValve_XV205 <= #0
#2 MixerOff:TON(IN: bFilling, PT: T#120m)
#3 AND(bFilling, NOT #2.Q)
#4 bSBRMixer <= #3
#5 AND(#2.Q, SBRLevelSensor_LSH200)
#6 bFillingDone <= #5
_END_CFC_
(* the same logic as Structured Text *)
bSBRValve_XV205 := bFilling AND SBRLevelSensor_LSH200;
MixerOff(IN := bFilling, PT := T#120m);
bSBRMixer := bFilling AND NOT MixerOff.Q;
bFillingDone := MixerOff.Q AND SBRLevelSensor_LSH200;
END_ACTION
ACTION Settle:
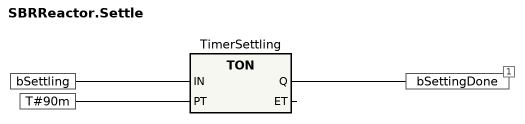
_CFC_ (* Continuous Function Chart, elements in execution order *)
#0 TimerSettling:TON(IN: bSettling, PT: T#90m)
#1 bSettingDone <= #0.Q
_END_CFC_
(* the same logic as Structured Text *)
TimerSettling(IN := bSettling, PT := T#90m);
bSettingDone := TimerSettling.Q;
END_ACTION

(* POU module/RangeBlock, ST *)
FUNCTION RangeBlock : BOOL
VAR_INPUT
	IN:REAL;
	LOWER : REAL;
	UPPER : REAL;
END_VAR
VAR
END_VAR
IF IN >= LOWER AND IN < UPPER THEN
	RangeBlock :=TRUE;
ELSE
	RangeBlock := FALSE;
END_IF
END_FUNCTION

(* POU SBR_REACTOR_1, CFC *)
PROGRAM SBR_REACTOR_1
VAR

	bDeSludge: BOOL;
	bBlower: BOOL;
	TimerStartBlower1: TON;
	TimerStartBlower2: TON;
	TimerStartBlower3: TON;
	tBlower1: fb_timer_on_off;
	tBlower2: fb_timer_on_off;
	tBlower3: fb_timer_on_off;



	SBR_A_1_SBRLevelSensor_LSH200 AT%I* : BOOL;
	SBR_A_1_DOSensor_DO201 AT%I* : INT;
	SBR_A_1_DecanterLevelSensorLow_Rx AT%I* : BOOL;
	SBR_A_1_DecanterLevelSensorHi_Rx AT%I* : BOOL;

	SBR_A_1_FowardDecant_XV26 AT%Q* : BOOL;
	SBR_A_1_ReverseDecant_XV26 AT%Q* : BOOL;
	SBR_A_1_BlowerValve_XV201 AT%Q* : BOOL;
	SBR_A_1_DeSludgeValve_XV241 AT%Q* : BOOL;
	SBR_A_1_SBRValve_XV205 AT%Q* : BOOL;
	SBR_A_1_SBRMixer_XV205  : BOOL;

	SBR_A_1_bEnable_SW : BOOL;
	SBR_A_1_Blower_B201 : BOOL;
	SBR_A_1_DesludgePump_P201 : BOOL;
	SBR_A_1_filling : BOOL;
	SBR_A_1_aeration : BOOL;
	SBR_A_1_settling : BOOL;
	SBR_A_1_decanting : BOOL;
	SBR_A_1_desludging : BOOL;
	SBR_A_1_SBRMixer_M200 : BOOL;
	SBR_A_1_warning_DONotInRange : BOOL;

	SBR_A_2_SBRLevelSensor_LSH200 AT%I* : BOOL;
	SBR_A_2_DOSensor_DO201 AT%I* : INT;
	SBR_A_2_DecanterLevelSensorLow_Rx AT%I* : BOOL;
	SBR_A_2_DecanterLevelSensorHi_Rx AT%I* : BOOL;

	SBR_A_2_FowardDecant_XV26 AT%Q* : BOOL;
	SBR_A_2_ReverseDecant_XV26 AT%Q* : BOOL;
	SBR_A_2_BlowerValve_XV201 AT%Q* : BOOL;
	SBR_A_2_DeSludgeValve_XV241 AT%Q* : BOOL;
	SBR_A_2_SBRValve_XV205 AT%Q* : BOOL;
	SBR_A_2_SBRMixer_XV205  : BOOL;

	SBR_A_2_bEnable_SW : BOOL;
	SBR_A_2_Blower_B201 : BOOL;
	SBR_A_2_DesludgePump_P201 : BOOL;
	SBR_A_2_filling : BOOL;
	SBR_A_2_aeration : BOOL;
	SBR_A_2_settling : BOOL;
	SBR_A_2_decanting : BOOL;
	SBR_A_2_desludging : BOOL;
	SBR_A_2_SBRMixer_M200 : BOOL;
	SBR_A_2_warning_DONotInRange : BOOL;

	SBR_A_3_SBRLevelSensor_LSH200 AT%I* : BOOL;
	SBR_A_3_DOSensor_DO201 AT%I* : INT;
	SBR_A_3_DecanterLevelSensorLow_Rx AT%I* : BOOL;
	SBR_A_3_DecanterLevelSensorHi_Rx AT%I* : BOOL;

	SBR_A_3_FowardDecant_XV26 AT%Q* : BOOL;
	SBR_A_3_ReverseDecant_XV26 AT%Q* : BOOL;
	SBR_A_3_BlowerValve_XV201 AT%Q* : BOOL;
	SBR_A_3_DeSludgeValve_XV241 AT%Q* : BOOL;
	SBR_A_3_SBRValve_XV205 AT%Q* : BOOL;
	SBR_A_3_SBRMixer_XV205  : BOOL;

	SBR_A_3_bEnable_SW : BOOL;
	SBR_A_3_Blower_B201 : BOOL;
	SBR_A_3_DesludgePump_P201 : BOOL;
	SBR_A_3_filling : BOOL;
	SBR_A_3_aeration : BOOL;
	SBR_A_3_settling : BOOL;
	SBR_A_3_decanting : BOOL;
	SBR_A_3_desludging : BOOL;
	SBR_A_3_SBRMixer_M200 : BOOL;
	SBR_A_3_warning_DONotInRange : BOOL;

	SBR_A_4_SBRLevelSensor_LSH200 AT%I* : BOOL;
	SBR_A_4_DOSensor_DO201 AT%I* : INT;
	SBR_A_4_DecanterLevelSensorLow_Rx AT%I* : BOOL;
	SBR_A_4_DecanterLevelSensorHi_Rx AT%I* : BOOL;

